KUKA KRL program: MyProgram_293().src

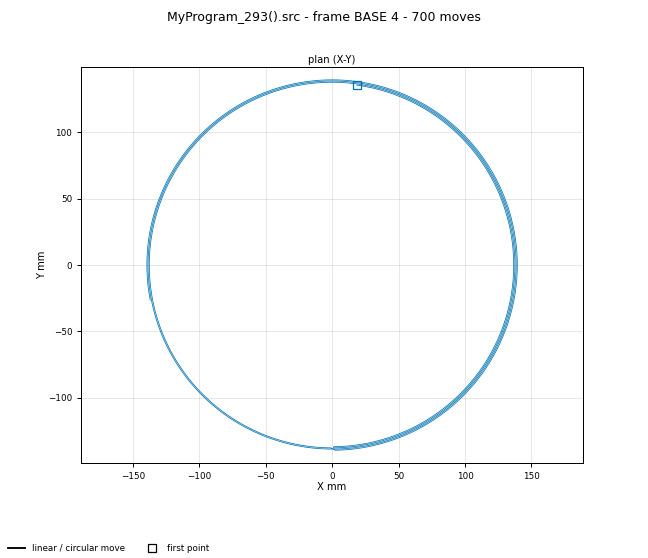
[picture p0: tool path of MyProgram_293().src in frame BASE 4, 700 of 700 moves have a stored position in this frame; points joined in program order, loops and branches not executed]
&ACCESS RVP
&REL 1
&PARAM TEMPLATE = C:\KRC\Roboter\Template\vorgabe
&PARAM EDITMASK = *
DEF MyProgram_293()
; ---- Setting reference (Base) ----
$BASE = BASE_DATA[4]

; --------------------------
; ---- Setting tool (TCP) ----
$TOOL = TOOL_DATA[3]
; --------------------------

$VEL.CP = VEL_APROX_PRINT
Startdeposition()
$VEL.CP = VEL_PRINT
LIN {X 18.5664,Y 135.4056,Z 177,A 82.6594,B 6.5518,C 0.1123,E1 6.5775,E2 369.6797} C_DIS
LIN {X 22.4593,Y 134.8123,Z 177,A 81.1585,B 6.5518,C 0.1109,E1 6.5816,E2 371.162} C_DIS
LIN {X 25.6947,Y 134.2332,Z 177,A 79.7863,B 6.5518,C 0.1116,E1 6.5854,E2 372.533} C_DIS
LIN {X 28.7602,Y 133.61,Z 177,A 78.4781,B 6.5518,C 0.1123,E1 6.589,E2 373.8405} C_DIS
LIN {X 32.2481,Y 132.8114,Z 177,A 76.9941,B 6.5518,C 0.1131,E1 6.593,E2 375.3222} C_DIS
LIN {X 35.7369,Y 131.9163,Z 177,A 75.4178,B 6.5518,C 0.1152,E1 6.5973,E2 376.9062} C_DIS
LIN {X 40.0506,Y 130.6702,Z 177,A 73.6118,B 6.5518,C 0.1156,E1 6.6021,E2 378.7026} C_DIS
LIN {X 43.4189,Y 129.5901,Z 177,A 72.1587,B 6.5517,C 0.1165,E1 6.6059,E2 380.1517} C_DIS
LIN {X 46.8464,Y 128.3916,Z 177,A 70.6202,B 6.5517,C 0.1182,E1 6.61,E2 381.6921} C_DIS
LIN {X 49.9108,Y 127.2313,Z 177,A 69.2422,B 6.5517,C 0.1197,E1 6.6136,E2 383.0704} C_DIS
LIN {X 52.8843,Y 126.0238,Z 177,A 67.9305,B 6.5517,C 0.1207,E1 6.6169,E2 384.3778} C_DIS
LIN {X 56.0642,Y 124.6418,Z 177,A 66.4902,B 6.5516,C 0.1222,E1 6.6206,E2 385.8164} C_DIS
LIN {X 59.3143,Y 123.1288,Z 177,A 64.9808,B 6.5516,C 0.1241,E1 6.6244,E2 387.3264} C_DIS
LIN {X 62.5726,Y 121.5062,Z 177,A 63.4613,B 6.5516,C 0.126,E1 6.6282,E2 388.8452} C_DIS
LIN {X 66.4914,Y 119.4079,Z 177,A 61.5636,B 6.5515,C 0.1291,E1 6.6329,E2 390.747} C_DIS
LIN {X 70.3636,Y 117.1681,Z 177,A 59.6863,B 6.5514,C 0.1319,E1 6.6374,E2 392.6246} C_DIS
LIN {X 74.1474,Y 114.8108,Z 177,A 57.8365,B 6.5514,C 0.1345,E1 6.6418,E2 394.4722} C_DIS
LIN {X 77.7972,Y 112.3696,Z 177,A 56.0558,B 6.5514,C 0.1365,E1 6.6459,E2 396.2457} C_DIS
LIN {X 81.159,Y 109.9661,Z 177,A 54.3535,B 6.5513,C 0.1389,E1 6.6497,E2 397.9445} C_DIS
LIN {X 84.4152,Y 107.4864,Z 177,A 52.6402,B 6.5512,C 0.1419,E1 6.6535,E2 399.6577} C_DIS
LIN {X 88.0221,Y 104.5534,Z 177,A 50.7109,B 6.5512,C 0.1452,E1 6.6576,E2 401.585} C_DIS
LIN {X 91.3809,Y 101.6309,Z 177,A 48.8831,B 6.5511,C 0.1481,E1 6.6614,E2 403.4084} C_DIS
LIN {X 95.3201,Y 97.9461,Z 177,A 46.6989,B 6.551,C 0.1513,E1 6.6659,E2 405.5837} C_DIS
LIN {X 98.313,Y 94.9411,Z 177,A 44.7068,B 6.5508,C 0.1584,E1 6.6698,E2 407.6024} C_DIS
LIN {X 100.5411,Y 92.5782,Z 177,A 43.7698,B 6.5509,C 0.1543,E1 6.6715,E2 408.4878} C_DIS
LIN {X 102.7371,Y 90.1358,Z 177,A 42.1809,B 6.5508,C 0.1608,E1 6.6745,E2 410.1031} C_DIS
LIN {X 105.6039,Y 86.7593,Z 177,A 40.2759,B 6.5506,C 0.1656,E1 6.6779,E2 412.0147} C_DIS
LIN {X 108.5925,Y 82.9874,Z 177,A 38.4354,B 6.5506,C 0.1672,E1 6.681,E2 413.8341} C_DIS
LIN {X 111.0305,Y 79.6965,Z 177,A 36.7303,B 6.5505,C 0.171,E1 6.6838,E2 415.5384} C_DIS
LIN {X 113.4927,Y 76.1495,Z 177,A 34.9398,B 6.5504,C 0.175,E1 6.6866,E2 417.3273} C_DIS
LIN {X 115.869,Y 72.4825,Z 177,A 33.1063,B 6.5503,C 0.1794,E1 6.6894,E2 419.1618} C_DIS
LIN {X 118.1937,Y 68.6259,Z 177,A 31.298,B 6.5502,C 0.1827,E1 6.692,E2 420.9611} C_DIS
LIN {X 120.235,Y 64.9838,Z 177,A 29.5546,B 6.5501,C 0.187,E1 6.6943,E2 422.7045} C_DIS
LIN {X 122.018,Y 61.5673,Z 177,A 28.0806,B 6.5501,C 0.1887,E1 6.6962,E2 424.1618} C_DIS
LIN {X 123.5453,Y 58.4425,Z 177,A 26.6295,B 6.5499,C 0.1923,E1 6.6979,E2 425.6128} C_DIS
LIN {X 125.2833,Y 54.6165,Z 177,A 24.7215,B 6.5497,C 0.1994,E1 6.7001,E2 427.5399} C_DIS
LIN {X 127.4324,Y 49.3935,Z 177,A 22.5717,B 6.5497,C 0.2019,E1 6.7023,E2 429.664} C_DIS
LIN {X 128.7184,Y 45.9402,Z 177,A 21.1087,B 6.5495,C 0.2047,E1 6.7037,E2 431.1179} C_DIS
LIN {X 129.7831,Y 42.8393,Z 177,A 19.728,B 6.5495,C 0.2085,E1 6.7049,E2 432.5002} C_DIS
LIN {X 130.8966,Y 39.3108,Z 177,A 18.2472,B 6.5493,C 0.2115,E1 6.7062,E2 433.9733} C_DIS
LIN {X 131.7436,Y 36.3672,Z 177,A 16.9687,B 6.5493,C 0.215,E1 6.7071,E2 435.2519} C_DIS
LIN {X 132.7743,Y 32.402,Z 177,A 15.2361,B 6.549,C 0.22,E1 6.7083,E2 436.9875} C_DIS
LIN {X 133.655,Y 28.5517,Z 177,A 13.6632,B 6.549,C 0.2232,E1 6.7093,E2 438.5512} C_DIS
LIN {X 134.3809,Y 24.9221,Z 177,A 12.0063,B 6.5487,C 0.2294,E1 6.7101,E2 440.2223} C_DIS
LIN {X 135.1025,Y 20.6444,Z 177,A 10.356,B 6.5487,C 0.2316,E1 6.7109,E2 441.853} C_DIS
LIN {X 135.6098,Y 17.0107,Z 177,A 8.7647,B 6.5485,C 0.2369,E1 6.7115,E2 443.4521} C_DIS
LIN {X 136.0754,Y 12.744,Z 177,A 7.0882,B 6.5483,C 0.2398,E1 6.7119,E2 445.1145} C_DIS
LIN {X 136.5806,Y 4.9707,Z 177,A 3.1417,B 6.5475,C 0.261,E1 6.7125,E2 449.1483} C_DIS
LIN {X 136.6684,Y -0.9178,Z 177,A 1.5135,B 6.5478,C 0.2535,E1 6.7125,E2 450.6738} C_DIS
LIN {X 136.5954,Y -4.5594,Z 177,A -0.5926,B 6.5473,C 0.2679,E1 6.7123,E2 452.8536} C_DIS
LIN {X 136.3436,Y -9.46,Z 177,A -2.4912,B 6.5471,C 0.2711,E1 6.712,E2 454.7342} C_DIS
LIN {X 135.9744,Y -13.7962,Z 177,A -3.8455,B 6.5473,C 0.2681,E1 6.7116,E2 456.0312} C_DIS
LIN {X 135.5357,Y -17.576,Z 177,A -5.43,B 6.5471,C 0.2725,E1 6.7111,E2 457.6157} C_DIS
LIN {X 134.9783,Y -21.4462,Z 177,A -7.0242,B 6.5469,C 0.2764,E1 6.7104,E2 459.2057} C_DIS
LIN {X 134.2054,Y -25.8402,Z 177,A -8.78,B 6.5468,C 0.2797,E1 6.7095,E2 460.9488} C_DIS
LIN {X 133.4372,Y -29.5604,Z 177,A -10.4906,B 6.5465,C 0.2862,E1 6.7085,E2 462.6757} C_DIS
LIN {X 132.2578,Y -34.4551,Z 177,A -12.5264,B 6.5463,C 0.2908,E1 6.7072,E2 464.704} C_DIS
LIN {X 131.2025,Y -38.2708,Z 177,A -14.1081,B 6.5461,C 0.2941,E1 6.706,E2 466.2773} C_DIS
LIN {X 130.0503,Y -42.022,Z 177,A -15.6724,B 6.5461,C 0.2972,E1 6.7047,E2 467.8329} C_DIS
LIN {X 128.5427,Y -46.4275,Z 177,A -17.6099,B 6.5458,C 0.3023,E1 6.7029,E2 469.7704} C_DIS
LIN {X 127.3413,Y -49.6278,Z 177,A -18.9635,B 6.5457,C 0.3048,E1 6.7015,E2 471.1152} C_DIS
LIN {X 125.9129,Y -53.1498,Z 177,A -20.5159,B 6.5455,C 0.3083,E1 6.6999,E2 472.664} C_DIS
LIN {X 124.6312,Y -56.088,Z 177,A -21.8391,B 6.5453,C 0.3115,E1 6.6984,E2 473.9858} C_DIS
LIN {X 123.3542,Y -58.8426,Z 177,A -23.2918,B 6.545,C 0.318,E1 6.6966,E2 475.4624} C_DIS
LIN {X 120.828,Y -63.8703,Z 177,A -25.421,B 6.545,C 0.3201,E1 6.694,E2 477.5647} C_DIS
LIN {X 118.8197,Y -67.5365,Z 177,A -27.2091,B 6.5447,C 0.3252,E1 6.6915,E2 479.3591} C_DIS
LIN {X 116.5896,Y -71.3171,Z 177,A -29.036,B 6.5445,C 0.3296,E1 6.6889,E2 481.1861} C_DIS
LIN {X 114.2108,Y -75.0675,Z 177,A -30.8592,B 6.5443,C 0.3335,E1 6.6861,E2 483.0061} C_DIS
LIN {X 111.7205,Y -78.726,Z 177,A -32.6652,B 6.5441,C 0.3371,E1 6.6833,E2 484.8075} C_DIS
LIN {X 109.1483,Y -82.2551,Z 177,A -34.483,B 6.5439,C 0.3412,E1 6.6802,E2 486.6255} C_DIS
LIN {X 106.402,Y -85.7779,Z 177,A -36.3143,B 6.5437,C 0.3448,E1 6.6771,E2 488.4533} C_DIS
LIN {X 103.4246,Y -89.3456,Z 177,A -38.2127,B 6.5435,C 0.3484,E1 6.6737,E2 490.3471} C_DIS
LIN {X 100.4923,Y -92.6313,Z 177,A -40.0388,B 6.5433,C 0.3521,E1 6.6702,E2 492.1724} C_DIS
LIN {X 97.385,Y -95.893,Z 177,A -41.8836,B 6.5431,C 0.3554,E1 6.6667,E2 494.0133} C_DIS
LIN {X 94.0387,Y -99.1762,Z 177,A -44.0328,B 6.5427,C 0.3625,E1 6.6623,E2 496.1876} C_DIS
LIN {X 91.5951,Y -101.4381,Z 177,A -45.4879,B 6.5425,C 0.3663,E1 6.6592,E2 497.6516} C_DIS
LIN {X 88.7953,Y -103.8978,Z 177,A -46.7251,B 6.5427,C 0.3639,E1 6.6567,E2 498.8488} C_DIS
LIN {X 85.4483,Y -106.6677,Z 177,A -48.5875,B 6.5424,C 0.368,E1 6.6527,E2 500.718} C_DIS
LIN {X 81.8828,Y -109.4283,Z 177,A -50.4029,B 6.5423,C 0.3702,E1 6.6487,E2 502.5255} C_DIS
LIN {X 78.4278,Y -111.9308,Z 177,A -52.2025,B 6.5421,C 0.3736,E1 6.6445,E2 504.3281} C_DIS
LIN {X 74.7223,Y -114.4375,Z 177,A -54.0556,B 6.542,C 0.3763,E1 6.6402,E2 506.1799} C_DIS
LIN {X 70.9075,Y -116.8393,Z 177,A -55.9071,B 6.5418,C 0.3787,E1 6.6359,E2 508.028} C_DIS
LIN {X 67.0797,Y -119.078,Z 177,A -57.7385,B 6.5417,C 0.3811,E1 6.6314,E2 509.8575} C_DIS
LIN {X 63.2452,Y -121.1563,Z 177,A -59.4788,B 6.5417,C 0.3823,E1 6.6272,E2 511.5879} C_DIS
LIN {X 60.1595,Y -122.7177,Z 177,A -60.9304,B 6.5415,C 0.3844,E1 6.6235,E2 513.0408} C_DIS
LIN {X 55.3417,Y -124.965,Z 177,A -63.1051,B 6.5414,C 0.3864,E1 6.618,E2 515.2104} C_DIS
LIN {X 46.6553,Y -128.4605,Z 177,A -66.795,B 6.5414,C 0.3873,E1 6.6085,E2 518.8732} C_DIS
LIN {X 43.9146,Y -129.425,Z 177,A -68.2318,B 6.541,C 0.392,E1 6.6046,E2 520.339} C_DIS
LIN {X 41.2908,Y -130.2839,Z 177,A -69.3344,B 6.541,C 0.3923,E1 6.6017,E2 521.4353} C_DIS
LIN {X 37.4387,Y -131.444,Z 177,A -71.1076,B 6.5408,C 0.3952,E1 6.5969,E2 523.2207} C_DIS
LIN {X 33.4016,Y -132.526,Z 177,A -72.7347,B 6.5408,C 0.3947,E1 6.5926,E2 524.833} C_DIS
LIN {X 30.3416,Y -133.2597,Z 177,A -74.0599,B 6.5408,C 0.3958,E1 6.589,E2 526.1597} C_DIS
LIN {X 27.0594,Y -133.9649,Z 177,A -75.4746,B 6.5408,C 0.3969,E1 6.5851,E2 527.5763} C_DIS
LIN {X 23.3736,Y -134.6587,Z 177,A -77.112,B 6.5406,C 0.3989,E1 6.5806,E2 529.223} C_DIS
LIN {X 16.7281,Y -135.6439,Z 177,A -79.715,B 6.5407,C 0.3972,E1 6.5735,E2 531.8004} C_DIS
LIN {X 12.2421,Y -136.1223,Z 177,A -82.1222,B 6.5402,C 0.4056,E1 6.5666,E2 534.2745} C_DIS
LIN {X 8.4372,Y -136.4098,Z 177,A -83.1352,B 6.5407,C 0.3974,E1 6.564,E2 535.2135} C_DIS
LIN {X 1.4274,Y -136.6648,Z 177,A -86.1789,B 6.5406,C 0.3996,E1 6.5554,E2 538.272} C_DIS
LIN {X 1.4274,Y -136.6648,Z 177,A -86.1789,B 6.5406,C 0.3996,E1 6.5554,E2 538.272} C_DIS
Enddeposition()
LIN {X 0.9977,Y -137.5702,Z 177,A -85.891,B 6.5463,C 0.3964,E1 6.5618,E2 537.955} C_DIS
Startdeposition()
$VEL.CP = VEL_PRINT
LIN {X 3.7285,Y -137.5249,Z 177,A -84.6313,B 6.5464,C 0.3944,E1 6.5654,E2 536.6789} C_DIS
LIN {X 6.8134,Y -137.4065,Z 177,A -83.3451,B 6.5464,C 0.3941,E1 6.569,E2 535.392} C_DIS
LIN {X 10.1117,Y -137.2032,Z 177,A -82.0399,B 6.5464,C 0.3947,E1 6.5726,E2 534.0952} C_DIS
LIN {X 13.0514,Y -136.9548,Z 177,A -80.7476,B 6.5465,C 0.3933,E1 6.5762,E2 532.794} C_DIS
LIN {X 16.3923,Y -136.5952,Z 177,A -79.4157,B 6.5465,C 0.3937,E1 6.5799,E2 531.4702} C_DIS
LIN {X 20.2553,Y -136.0783,Z 177,A -77.7612,B 6.5465,C 0.3924,E1 6.5845,E2 529.8107} C_DIS
LIN {X 23.4383,Y -135.5663,Z 177,A -76.4224,B 6.5466,C 0.3916,E1 6.5882,E2 528.4716} C_DIS
LIN {X 26.6321,Y -134.9752,Z 177,A -75.0021,B 6.5467,C 0.3897,E1 6.5921,E2 527.0416} C_DIS
LIN {X 30.34,Y -134.1882,Z 177,A -73.4718,B 6.5467,C 0.3893,E1 6.5963,E2 525.5165} C_DIS
LIN {X 34.6459,Y -133.1436,Z 177,A -71.6655,B 6.5467,C 0.3884,E1 6.6011,E2 523.7142} C_DIS
LIN {X 37.8556,Y -132.2669,Z 177,A -70.2873,B 6.5469,C 0.3873,E1 6.6048,E2 522.3361} C_DIS
LIN {X 41.2103,Y -131.2594,Z 177,A -68.8943,B 6.5469,C 0.387,E1 6.6085,E2 520.9506} C_DIS
LIN {X 44.2654,Y -130.2618,Z 177,A -67.4751,B 6.547,C 0.3843,E1 6.6123,E2 519.5199} C_DIS
LIN {X 47.4593,Y -129.1324,Z 177,A -66.1069,B 6.547,C 0.3835,E1 6.6159,E2 518.1562} C_DIS
LIN {X 50.6416,Y -127.918,Z 177,A -64.6992,B 6.5472,C 0.382,E1 6.6196,E2 516.7489} C_DIS
LIN {X 54.2347,Y -126.4341,Z 177,A -63.1019,B 6.5472,C 0.3804,E1 6.6237,E2 515.1531} C_DIS
LIN {X 56.9581,Y -125.2331,Z 177,A -61.8648,B 6.5473,C 0.3788,E1 6.6268,E2 513.9156} C_DIS
LIN {X 60.0858,Y -123.7629,Z 177,A -60.439,B 6.5474,C 0.3771,E1 6.6304,E2 512.4904} C_DIS
LIN {X 63.1886,Y -122.2079,Z 177,A -58.8981,B 6.5477,C 0.3735,E1 6.6343,E2 510.9358} C_DIS
LIN {X 67.027,Y -120.1456,Z 177,A -57.1262,B 6.5477,C 0.3716,E1 6.6386,E2 509.168} C_DIS
LIN {X 70.8146,Y -117.9528,Z 177,A -55.3047,B 6.5479,C 0.3688,E1 6.643,E2 507.3453} C_DIS
LIN {X 74.5451,Y -115.6313,Z 177,A -53.4961,B 6.5481,C 0.3661,E1 6.6473,E2 505.5379} C_DIS
LIN {X 78.2897,Y -113.1292,Z 177,A -51.6664,B 6.5482,C 0.3637,E1 6.6515,E2 503.7126} C_DIS
LIN {X 81.8087,Y -110.6115,Z 177,A -49.8837,B 6.5484,C 0.3608,E1 6.6555,E2 501.9309} C_DIS
LIN {X 85.3293,Y -107.9189,Z 177,A -48.04,B 6.5485,C 0.3575,E1 6.6596,E2 500.0858} C_DIS
LIN {X 88.7677,Y -105.1088,Z 177,A -46.24,B 6.5487,C 0.3548,E1 6.6634,E2 498.2906} C_DIS
LIN {X 92.1181,Y -102.1852,Z 177,A -44.3969,B 6.5489,C 0.3512,E1 6.6673,E2 496.4469} C_DIS
LIN {X 95.3794,Y -99.1481,Z 177,A -42.571,B 6.5491,C 0.348,E1 6.671,E2 494.6233} C_DIS
LIN {X 98.533,Y -96.0147,Z 177,A -40.7667,B 6.5492,C 0.3449,E1 6.6745,E2 492.8235} C_DIS
LIN {X 101.5873,Y -92.7771,Z 177,A -38.9249,B 6.5494,C 0.341,E1 6.678,E2 490.9815} C_DIS
LIN {X 104.5331,Y -89.445,Z 177,A -37.1234,B 6.5496,C 0.3378,E1 6.6813,E2 489.1849} C_DIS
LIN {X 107.3661,Y -86.0237,Z 177,A -35.3063,B 6.5498,C 0.3341,E1 6.6845,E2 487.3703} C_DIS
LIN {X 110.0826,Y -82.5191,Z 177,A -33.4933,B 6.55,C 0.3304,E1 6.6876,E2 485.56} C_DIS
LIN {X 112.6788,Y -78.937,Z 177,A -31.6667,B 6.5502,C 0.3263,E1 6.6905,E2 483.7337} C_DIS
LIN {X 115.1518,Y -75.2838,Z 177,A -29.8604,B 6.5504,C 0.3223,E1 6.6933,E2 481.9297} C_DIS
LIN {X 117.4987,Y -71.5655,Z 177,A -28.0881,B 6.5505,C 0.3188,E1 6.6959,E2 480.1634} C_DIS
LIN {X 119.7174,Y -67.7888,Z 177,A -26.2978,B 6.5507,C 0.3148,E1 6.6984,E2 478.3757} C_DIS
LIN {X 121.3987,Y -64.7296,Z 177,A -24.9613,B 6.5508,C 0.3131,E1 6.7002,E2 477.053} C_DIS
LIN {X 122.996,Y -61.6405,Z 177,A -23.5235,B 6.551,C 0.3096,E1 6.702,E2 475.6152} C_DIS
LIN {X 124.6916,Y -58.1293,Z 177,A -22.1099,B 6.551,C 0.309,E1 6.7036,E2 474.2272} C_DIS
LIN {X 126.1301,Y -54.9379,Z 177,A -20.7016,B 6.5511,C 0.306,E1 6.7052,E2 472.8239} C_DIS
LIN {X 127.2787,Y -52.2273,Z 177,A -19.3258,B 6.5514,C 0.3001,E1 6.7067,E2 471.4278} C_DIS
LIN {X 128.5358,Y -49.0521,Z 177,A -17.9343,B 6.5516,C 0.2968,E1 6.7081,E2 470.0389} C_DIS
LIN {X 129.7078,Y -45.8636,Z 177,A -16.5505,B 6.5517,C 0.2935,E1 6.7095,E2 468.6577} C_DIS
LIN {X 130.7947,Y -42.6651,Z 177,A -15.1743,B 6.5519,C 0.2902,E1 6.7107,E2 467.2843} C_DIS
LIN {X 131.7972,Y -39.4598,Z 177,A -13.8072,B 6.552,C 0.2869,E1 6.7118,E2 465.9199} C_DIS
LIN {X 132.7157,Y -36.2508,Z 177,A -12.4483,B 6.5521,C 0.2836,E1 6.7128,E2 464.5637} C_DIS
LIN {X 133.5509,Y -33.0413,Z 177,A -11.0985,B 6.5523,C 0.2802,E1 6.7137,E2 463.2167} C_DIS
LIN {X 134.3357,Y -29.6861,Z 177,A -9.6225,B 6.5525,C 0.2755,E1 6.7146,E2 461.7341} C_DIS
LIN {X 134.9752,Y -26.6321,Z 177,A -8.3075,B 6.5527,C 0.2715,E1 6.7154,E2 460.416} C_DIS
LIN {X 135.5663,Y -23.4383,Z 177,A -7.1048,B 6.5527,C 0.2704,E1 6.7159,E2 459.2314} C_DIS
LIN {X 136.0783,Y -20.2553,Z 177,A -5.7931,B 6.5528,C 0.2671,E1 6.7165,E2 457.9225} C_DIS
LIN {X 136.579,Y -16.528,Z 177,A -4.4655,B 6.5528,C 0.2669,E1 6.717,E2 456.624} C_DIS
LIN {X 136.8703,Y -13.932,Z 177,A -3.201,B 6.5531,C 0.2606,E1 6.7174,E2 455.3361} C_DIS
LIN {X 137.1532,Y -10.7967,Z 177,A -1.9207,B 6.5532,C 0.2574,E1 6.7176,E2 454.0586} C_DIS
LIN {X 137.3629,Y -7.6821,Z 177,A -0.6516,B 6.5533,C 0.2543,E1 6.7179,E2 452.7924} C_DIS
LIN {X 137.5009,Y -4.5903,Z 177,A 0.7505,B 6.5536,C 0.2485,E1 6.718,E2 451.3747} C_DIS
LIN {X 137.5691,Y -1.5235,Z 177,A 1.8807,B 6.5536,C 0.2475,E1 6.718,E2 450.2623} C_DIS
LIN {X 137.5691,Y 1.5235,Z 177,A 3.0967,B 6.5537,C 0.2448,E1 6.718,E2 449.0521} C_DIS
LIN {X 137.5009,Y 4.5903,Z 177,A 4.3491,B 6.5538,C 0.2416,E1 6.718,E2 447.8018} C_DIS
LIN {X 137.3629,Y 7.6821,Z 177,A 5.6126,B 6.5539,C 0.2383,E1 6.7178,E2 446.5406} C_DIS
LIN {X 137.1532,Y 10.7967,Z 177,A 6.9567,B 6.5541,C 0.2339,E1 6.7175,E2 445.1898} C_DIS
LIN {X 136.8703,Y 13.932,Z 177,A 8.172,B 6.5541,C 0.2318,E1 6.7172,E2 443.9857} C_DIS
LIN {X 136.5125,Y 17.0857,Z 177,A 9.4679,B 6.5543,C 0.2285,E1 6.7167,E2 442.6922} C_DIS
LIN {X 136.0783,Y 20.2553,Z 177,A 10.7736,B 6.5544,C 0.2252,E1 6.7162,E2 441.3889} C_DIS
LIN {X 135.4654,Y 24.0017,Z 177,A 12.2904,B 6.5545,C 0.2219,E1 6.7155,E2 439.879} C_DIS
LIN {X 134.9719,Y 26.6483,Z 177,A 13.4166,B 6.5546,C 0.2186,E1 6.7149,E2 438.7514} C_DIS
LIN {X 134.3038,Y 29.834,Z 177,A 14.7514,B 6.5547,C 0.2152,E1 6.7141,E2 437.4184} C_DIS
LIN {X 133.5509,Y 33.0413,Z 177,A 16.1839,B 6.5549,C 0.2104,E1 6.7132,E2 435.9772} C_DIS
LIN {X 132.6126,Y 36.6192,Z 177,A 17.6102,B 6.5549,C 0.2081,E1 6.7121,E2 434.5644} C_DIS
LIN {X 131.7972,Y 39.4598,Z 177,A 18.8138,B 6.5551,C 0.2052,E1 6.7112,E2 433.3635} C_DIS
LIN {X 130.6278,Y 43.1663,Z 177,A 20.3612,B 6.5551,C 0.202,E1 6.7099,E2 431.8239} C_DIS
LIN {X 129.6113,Y 46.1312,Z 177,A 21.5781,B 6.5552,C 0.2001,E1 6.7088,E2 430.6176} C_DIS
LIN {X 128.5358,Y 49.0521,Z 177,A 22.9527,B 6.5554,C 0.1952,E1 6.7074,E2 429.2322} C_DIS
LIN {X 127.2787,Y 52.2273,Z 177,A 24.4355,B 6.5555,C 0.1904,E1 6.7059,E2 427.7409} C_DIS
LIN {X 125.9363,Y 55.386,Z 177,A 25.8381,B 6.5555,C 0.1871,E1 6.7043,E2 426.341} C_DIS
LIN {X 124.5087,Y 58.5249,Z 177,A 27.1595,B 6.5556,C 0.1854,E1 6.7028,E2 425.0333} C_DIS
LIN {X 122.996,Y 61.6405,Z 177,A 28.6123,B 6.5558,C 0.1815,E1 6.701,E2 423.5784} C_DIS
LIN {X 121.059,Y 65.362,Z 177,A 30.3076,B 6.5558,C 0.178,E1 6.6988,E2 421.8888} C_DIS
LIN {X 119.0914,Y 68.8812,Z 177,A 32.0128,B 6.556,C 0.1734,E1 6.6964,E2 420.1795} C_DIS
LIN {X 116.7791,Y 72.7325,Z 177,A 33.8466,B 6.556,C 0.1695,E1 6.6937,E2 418.3495} C_DIS
LIN {X 114.3926,Y 76.4311,Z 177,A 35.6313,B 6.5562,C 0.1659,E1 6.691,E2 416.5701} C_DIS
LIN {X 111.8808,Y 80.0628,Z 177,A 37.4386,B 6.5562,C 0.1622,E1 6.6881,E2 414.766} C_DIS
LIN {X 109.3123,Y 83.5356,Z 177,A 39.2275,B 6.5564,C 0.1582,E1 6.6851,E2 412.9778} C_DIS
LIN {X 106.4935,Y 87.1006,Z 177,A 41.0684,B 6.5564,C 0.1549,E1 6.6819,E2 411.1427} C_DIS
LIN {X 103.5973,Y 90.5261,Z 177,A 42.8987,B 6.5565,C 0.1515,E1 6.6786,E2 409.3166} C_DIS
LIN {X 100.6447,Y 93.7977,Z 177,A 44.7123,B 6.5565,C 0.148,E1 6.6751,E2 407.5052} C_DIS
LIN {X 97.5157,Y 97.0468,Z 177,A 46.5511,B 6.5567,C 0.1448,E1 6.6716,E2 405.6709} C_DIS
LIN {X 94.447,Y 100.0357,Z 177,A 48.339,B 6.5567,C 0.1412,E1 6.668,E2 403.8821} C_DIS
LIN {X 91.0815,Y 103.1093,Z 177,A 50.1885,B 6.5568,C 0.1383,E1 6.6641,E2 402.0383} C_DIS
LIN {X 87.7864,Y 105.9289,Z 177,A 51.9892,B 6.5568,C 0.1351,E1 6.6603,E2 400.238} C_DIS
LIN {X 84.2772,Y 108.7416,Z 177,A 53.8245,B 6.5569,C 0.1324,E1 6.6563,E2 398.4071} C_DIS
LIN {X 80.6195,Y 111.4804,Z 177,A 55.6771,B 6.5569,C 0.13,E1 6.6521,E2 396.5606} C_DIS
LIN {X 77.0741,Y 113.9603,Z 177,A 57.4712,B 6.557,C 0.1272,E1 6.648,E2 394.7673} C_DIS
LIN {X 73.3868,Y 116.3691,Z 177,A 59.2823,B 6.557,C 0.1247,E1 6.6437,E2 392.959} C_DIS
LIN {X 69.7298,Y 118.5966,Z 177,A 61.0643,B 6.5571,C 0.1221,E1 6.6395,E2 391.1772} C_DIS
LIN {X 65.9269,Y 120.7519,Z 177,A 62.8145,B 6.5571,C 0.1206,E1 6.6352,E2 389.4357} C_DIS
LIN {X 63.1886,Y 122.2079,Z 177,A 64.1332,B 6.5571,C 0.1185,E1 6.6319,E2 388.1137} C_DIS
LIN {X 60.0858,Y 123.7629,Z 177,A 65.4966,B 6.5571,C 0.1179,E1 6.6285,E2 386.7605} C_DIS
LIN {X 56.9581,Y 125.2331,Z 177,A 67.053,B 6.5573,C 0.1144,E1 6.6246,E2 385.1897} C_DIS
LIN {X 53.4574,Y 126.765,Z 177,A 68.3572,B 6.5573,C 0.117,E1 6.6213,E2 383.9212} C_DIS
LIN {X 50.6416,Y 127.918,Z 177,A 69.7521,B 6.5573,C 0.1137,E1 6.6177,E2 382.5107} C_DIS
LIN {X 47.4593,Y 129.1324,Z 177,A 71.2995,B 6.5573,C 0.1102,E1 6.6136,E2 380.9475} C_DIS
LIN {X 43.8871,Y 130.3878,Z 177,A 72.6905,B 6.5573,C 0.1116,E1 6.6099,E2 379.5797} C_DIS
LIN {X 40.8564,Y 131.3697,Z 177,A 73.9579,B 6.5573,C 0.1113,E1 6.6066,E2 378.32} C_DIS
LIN {X 37.8556,Y 132.2669,Z 177,A 75.332,B 6.5573,C 0.1092,E1 6.6029,E2 376.9376} C_DIS
LIN {X 34.3144,Y 133.2278,Z 177,A 76.7233,B 6.5573,C 0.1101,E1 6.5992,E2 375.5634} C_DIS
LIN {X 31.4372,Y 133.9376,Z 177,A 78.1706,B 6.5573,C 0.1061,E1 6.5952,E2 374.0902} C_DIS
LIN {X 28.2322,Y 134.6496,Z 177,A 79.4332,B 6.5573,C 0.1068,E1 6.5918,E2 372.8408} C_DIS
LIN {X 24.5213,Y 135.3725,Z 177,A 80.9678,B 6.5573,C 0.1065,E1 6.5876,E2 371.3115} C_DIS
LIN {X 21.2848,Y 135.9189,Z 177,A 82.3883,B 6.5574,C 0.1051,E1 6.5836,E2 369.8849} C_DIS
LIN {X 17.0857,Y 136.5125,Z 177,A 84.1163,B 6.5574,C 0.105,E1 6.5789,E2 368.1623} C_DIS
LIN {X 13.932,Y 136.8703,Z 177,A 85.4324,B 6.5574,C 0.1046,E1 6.5752,E2 366.8474} C_DIS
LIN {X 10.7967,Y 137.1532,Z 177,A 86.7385,B 6.5574,C 0.1043,E1 6.5716,E2 365.5424} C_DIS
LIN {X 7.6821,Y 137.3629,Z 177,A 88.0337,B 6.5574,C 0.1042,E1 6.568,E2 364.2482} C_DIS
LIN {X 4.5903,Y 137.5009,Z 177,A 89.3189,B 6.5574,C 0.1041,E1 6.5644,E2 362.9641} C_DIS
LIN {X 1.5235,Y 137.5691,Z 177,A 90.5934,B 6.5574,C 0.1041,E1 6.5608,E2 361.6905} C_DIS
LIN {X -1.5235,Y 137.5691,Z 177,A 91.8634,B 6.5574,C 0.104,E1 6.5573,E2 360.4209} C_DIS
LIN {X -4.5903,Y 137.5009,Z 177,A 93.2485,B 6.5574,C 0.1026,E1 6.5534,E2 359.0231} C_DIS
LIN {X -7.6821,Y 137.3629,Z 177,A 94.4372,B 6.5574,C 0.1041,E1 6.5501,E2 357.8475} C_DIS
LIN {X -10.7967,Y 137.1532,Z 177,A 95.7417,B 6.5574,C 0.1043,E1 6.5465,E2 356.5431} C_DIS
LIN {X -13.932,Y 136.8703,Z 177,A 97.0578,B 6.5574,C 0.1046,E1 6.5428,E2 355.227} C_DIS
LIN {X -17.0857,Y 136.5125,Z 177,A 98.5408,B 6.5574,C 0.1028,E1 6.5386,E2 353.7248} C_DIS
LIN {X -20.2553,Y 136.0783,Z 177,A 99.7241,B 6.5574,C 0.1054,E1 6.5354,E2 352.5607} C_DIS
LIN {X -23.4383,Y 135.5663,Z 177,A 101.0738,B 6.5574,C 0.1059,E1 6.5317,E2 351.2108} C_DIS
LIN {X -26.6321,Y 134.9752,Z 177,A 102.4344,B 6.5574,C 0.1065,E1 6.528,E2 349.8501} C_DIS
LIN {X -29.834,Y 134.3038,Z 177,A 103.9,B 6.5574,C 0.1059,E1 6.5239,E2 348.3726} C_DIS
LIN {X -33.162,Y 133.5203,Z 177,A 105.1919,B 6.5574,C 0.1086,E1 6.5205,E2 347.0978} C_DIS
LIN {X -36.2508,Y 132.7157,Z 177,A 106.5772,B 6.5574,C 0.1088,E1 6.5167,E2 345.7065} C_DIS
LIN {X -39.4598,Y 131.7972,Z 177,A 108.0792,B 6.5574,C 0.1085,E1 6.5127,E2 344.1916} C_DIS
LIN {X -43.2174,Y 130.6108,Z 177,A 109.4149,B 6.5573,C 0.1139,E1 6.5092,E2 342.8946} C_DIS
LIN {X -45.8636,Y 129.7078,Z 177,A 110.8068,B 6.5573,C 0.112,E1 6.5055,E2 341.4755} C_DIS
LIN {X -49.5378,Y 128.347,Z 177,A 112.2585,B 6.5573,C 0.116,E1 6.5017,E2 340.0471} C_DIS
LIN {X -52.2273,Y 127.2787,Z 177,A 113.6702,B 6.5573,C 0.1146,E1 6.498,E2 338.6108} C_DIS
LIN {X -55.386,Y 125.9363,Z 177,A 115.2271,B 6.5573,C 0.1146,E1 6.494,E2 337.0392} C_DIS
LIN {X -58.7225,Y 124.4143,Z 177,A 116.5749,B 6.5572,C 0.1187,E1 6.4906,E2 335.7147} C_DIS
LIN {X -61.6405,Y 122.996,Z 177,A 118.0229,B 6.5572,C 0.1191,E1 6.487,E2 334.2559} C_DIS
LIN {X -65.1602,Y 121.1674,Z 177,A 119.7489,B 6.5572,C 0.1204,E1 6.4827,E2 332.5219} C_DIS
LIN {X -68.8897,Y 119.0865,Z 177,A 121.5678,B 6.5572,C 0.1224,E1 6.4783,E2 330.6994} C_DIS
LIN {X -72.7325,Y 116.7791,Z 177,A 123.4391,B 6.5571,C 0.1251,E1 6.4738,E2 328.829} C_DIS
LIN {X -76.4311,Y 114.3926,Z 177,A 125.2962,B 6.5571,C 0.1277,E1 6.4695,E2 326.9704} C_DIS
LIN {X -80.0628,Y 111.8808,Z 177,A 127.1602,B 6.557,C 0.1304,E1 6.4652,E2 325.1049} C_DIS
LIN {X -83.5356,Y 109.3123,Z 177,A 129.0056,B 6.557,C 0.1329,E1 6.4611,E2 323.2553} C_DIS
LIN {X -87.1006,Y 106.4935,Z 177,A 130.9105,B 6.5568,C 0.1361,E1 6.4569,E2 321.3504} C_DIS
LIN {X -90.5652,Y 103.5632,Z 177,A 132.8063,B 6.5568,C 0.1396,E1 6.4529,E2 319.4555} C_DIS
LIN {X -93.7977,Y 100.6447,Z 177,A 134.665,B 6.5568,C 0.1426,E1 6.4491,E2 317.5929} C_DIS
LIN {X -97.0046,Y 97.5576,Z 177,A 136.5483,B 6.5566,C 0.1459,E1 6.4453,E2 315.7076} C_DIS
LIN {X -100.0357,Y 94.447,Z 177,A 138.4079,B 6.5566,C 0.149,E1 6.4417,E2 313.8432} C_DIS
LIN {X -103.1093,Y 91.0815,Z 177,A 140.3166,B 6.5565,C 0.153,E1 6.4382,E2 311.935} C_DIS
LIN {X -105.9872,Y 87.7159,Z 177,A 142.2105,B 6.5564,C 0.1564,E1 6.4348,E2 310.0366} C_DIS
LIN {X -108.7846,Y 84.2216,Z 177,A 144.0854,B 6.5563,C 0.1605,E1 6.4315,E2 308.162} C_DIS
LIN {X -111.3637,Y 80.7806,Z 177,A 145.9335,B 6.5563,C 0.164,E1 6.4284,E2 306.3085} C_DIS
LIN {X -113.9603,Y 77.0741,Z 177,A 147.8313,B 6.5561,C 0.1683,E1 6.4254,E2 304.4107} C_DIS
LIN {X -116.3691,Y 73.3868,Z 177,A 149.6996,B 6.556,C 0.1723,E1 6.4226,E2 302.54} C_DIS
LIN {X -118.5966,Y 69.7298,Z 177,A 151.5374,B 6.5559,C 0.1761,E1 6.42,E2 300.697} C_DIS
LIN {X -120.7519,Y 65.9269,Z 177,A 153.2175,B 6.5557,C 0.1823,E1 6.4177,E2 299.0361} C_DIS
LIN {X -122.2079,Y 63.1886,Z 177,A 154.6326,B 6.5557,C 0.1841,E1 6.4159,E2 297.6068} C_DIS
LIN {X -123.7629,Y 60.0858,Z 177,A 156.1063,B 6.5556,C 0.1875,E1 6.414,E2 296.1309} C_DIS
LIN {X -125.3395,Y 56.7204,Z 177,A 157.5862,B 6.5554,C 0.1924,E1 6.4123,E2 294.6609} C_DIS
LIN {X -126.6787,Y 53.6641,Z 177,A 159.0427,B 6.5554,C 0.1953,E1 6.4107,E2 293.1973} C_DIS
LIN {X -127.918,Y 50.6416,Z 177,A 160.6076,B 6.5554,C 0.1966,E1 6.409,E2 291.6081} C_DIS
LIN {X -129.1324,Y 47.4593,Z 177,A 161.9374,B 6.5552,C 0.2014,E1 6.4078,E2 290.2908} C_DIS
LIN {X -130.2618,Y 44.2654,Z 177,A 163.3767,B 6.5551,C 0.2049,E1 6.4064,E2 288.8493} C_DIS
LIN {X -131.4648,Y 40.5458,Z 177,A 164.9089,B 6.5549,C 0.2104,E1 6.4052,E2 287.3304} C_DIS
LIN {X -132.2669,Y 37.8556,Z 177,A 166.2316,B 6.5549,C 0.2119,E1 6.4041,E2 285.9896} C_DIS
LIN {X -133.1436,Y 34.6459,Z 177,A 167.6459,B 6.5547,C 0.2155,E1 6.4031,E2 284.573} C_DIS
LIN {X -133.9376,Y 31.4372,Z 177,A 169.1959,B 6.5547,C 0.2173,E1 6.4021,E2 283.0024} C_DIS
LIN {X -134.6496,Y 28.2322,Z 177,A 170.4466,B 6.5545,C 0.2225,E1 6.4013,E2 281.7677} C_DIS
LIN {X -135.2807,Y 25.034,Z 177,A 171.8326,B 6.5544,C 0.226,E1 6.4006,E2 280.3793} C_DIS
LIN {X -135.9049,Y 21.3746,Z 177,A 173.4431,B 6.5542,C 0.2297,E1 6.3999,E2 278.7619} C_DIS
LIN {X -136.349,Y 18.3326,Z 177,A 174.6502,B 6.5541,C 0.2341,E1 6.3994,E2 277.5652} C_DIS
LIN {X -136.7646,Y 14.9136,Z 177,A 175.9567,B 6.5539,C 0.2396,E1 6.399,E2 276.276} C_DIS
LIN {X -137.021,Y 12.3619,Z 177,A 177.2728,B 6.5539,C 0.2399,E1 6.3986,E2 274.9297} C_DIS
LIN {X -137.2671,Y 9.2367,Z 177,A 178.6057,B 6.5538,C 0.2433,E1 6.3984,E2 273.5945} C_DIS
LIN {X -137.4619,Y 5.5906,Z 177,A -179.7872,B 6.5536,C 0.2467,E1 6.3982,E2 271.9777} C_DIS
LIN {X -137.562,Y 1.9459,Z 177,A -178.2219,B 6.5535,C 0.2505,E1 6.3981,E2 270.4077} C_DIS
LIN {X -137.5691,Y -1.5235,Z 177,A -176.8133,B 6.5533,C 0.2551,E1 6.3981,E2 269.0049} C_DIS
LIN {X -137.5009,Y -4.5903,Z 177,A -175.5038,B 6.5532,C 0.2584,E1 6.3981,E2 267.6924} C_DIS
LIN {X -137.3466,Y -7.9456,Z 177,A -174.0181,B 6.5531,C 0.2614,E1 6.3984,E2 266.1968} C_DIS
LIN {X -137.0951,Y -11.4841,Z 177,A -172.5555,B 6.5529,C 0.2658,E1 6.3987,E2 264.7373} C_DIS
LIN {X -136.7008,Y -15.5067,Z 177,A -170.8319,B 6.5527,C 0.2701,E1 6.3992,E2 263.0099} C_DIS
LIN {X -136.305,Y -18.6686,Z 177,A -169.3401,B 6.5527,C 0.272,E1 6.3998,E2 261.4982} C_DIS
LIN {X -135.8097,Y -21.9792,Z 177,A -168.0541,B 6.5524,C 0.2771,E1 6.4003,E2 260.2269} C_DIS
LIN {X -135.2666,Y -25.1075,Z 177,A -166.7189,B 6.5523,C 0.2807,E1 6.401,E2 258.891} C_DIS
LIN {X -134.6381,Y -28.2854,Z 177,A -165.2941,B 6.5521,C 0.2836,E1 6.4018,E2 257.4576} C_DIS
LIN {X -133.9031,Y -31.5804,Z 177,A -163.9253,B 6.552,C 0.2879,E1 6.4026,E2 256.0944} C_DIS
LIN {X -133.1436,Y -34.6459,Z 177,A -162.5234,B 6.5518,C 0.2906,E1 6.4036,E2 254.6825} C_DIS
LIN {X -132.2669,Y -37.8556,Z 177,A -161.1054,B 6.5517,C 0.294,E1 6.4047,E2 253.2613} C_DIS
LIN {X -131.1661,Y -41.5025,Z 177,A -159.4634,B 6.5515,C 0.2976,E1 6.406,E2 251.6132} C_DIS
LIN {X -130.2618,Y -44.2654,Z 177,A -158.2363,B 6.5514,C 0.3007,E1 6.4071,E2 250.3848} C_DIS
LIN {X -129.1324,Y -47.4593,Z 177,A -156.8016,B 6.5512,C 0.3042,E1 6.4085,E2 248.948} C_DIS
LIN {X -127.918,Y -50.6416,Z 177,A -155.3516,B 6.5511,C 0.3076,E1 6.41,E2 247.4949} C_DIS
LIN {X -126.6136,Y -53.8195,Z 177,A -153.7817,B 6.551,C 0.3097,E1 6.4117,E2 245.9079} C_DIS
LIN {X -125.2331,Y -56.9581,Z 177,A -152.4309,B 6.5508,C 0.3143,E1 6.4132,E2 244.5678} C_DIS
LIN {X -123.6546,Y -60.3054,Z 177,A -150.8304,B 6.5506,C 0.3175,E1 6.4151,E2 242.9606} C_DIS
LIN {X -122.1878,Y -63.2268,Z 177,A -149.3733,B 6.5505,C 0.3198,E1 6.417,E2 241.4919} C_DIS
LIN {X -120.1456,Y -67.027,Z 177,A -147.5445,B 6.5503,C 0.3239,E1 6.4195,E2 239.66} C_DIS
LIN {X -117.9528,Y -70.8146,Z 177,A -145.6656,B 6.5501,C 0.3276,E1 6.4222,E2 237.7747} C_DIS
LIN {X -115.6313,Y -74.5451,Z 177,A -143.7998,B 6.5499,C 0.3315,E1 6.425,E2 235.9051} C_DIS
LIN {X -113.1833,Y -78.2119,Z 177,A -141.9285,B 6.5497,C 0.3353,E1 6.4279,E2 234.0301} C_DIS
LIN {X -110.6081,Y -81.8133,Z 177,A -140.0715,B 6.5495,C 0.3393,E1 6.431,E2 232.1721} C_DIS
LIN {X -107.9189,Y -85.3293,Z 177,A -138.1739,B 6.5493,C 0.3427,E1 6.4342,E2 230.2682} C_DIS
LIN {X -105.1088,Y -88.7677,Z 177,A -136.3063,B 6.5491,C 0.3465,E1 6.4376,E2 228.3989} C_DIS
LIN {X -102.1852,Y -92.1181,Z 177,A -134.4099,B 6.549,C 0.3498,E1 6.4411,E2 226.4973} C_DIS
LIN {X -99.1003,Y -95.4288,Z 177,A -132.5137,B 6.5488,C 0.3534,E1 6.4447,E2 224.6002} C_DIS
LIN {X -96.0147,Y -98.533,Z 177,A -130.6639,B 6.5486,C 0.3566,E1 6.4484,E2 222.7473} C_DIS
LIN {X -92.7771,Y -101.5873,Z 177,A -128.7634,B 6.5484,C 0.3595,E1 6.4523,E2 220.8411} C_DIS
LIN {X -89.445,Y -104.5331,Z 177,A -126.9049,B 6.5483,C 0.3627,E1 6.4562,E2 218.9821} C_DIS
LIN {X -86.0237,Y -107.3661,Z 177,A -125.0304,B 6.5481,C 0.3656,E1 6.4603,E2 217.1048} C_DIS
LIN {X -82.5191,Y -110.0826,Z 177,A -123.1606,B 6.5479,C 0.3683,E1 6.4645,E2 215.2323} C_DIS
LIN {X -78.937,Y -112.6788,Z 177,A -121.2772,B 6.5479,C 0.3707,E1 6.4688,E2 213.3437} C_DIS
LIN {X -75.2838,Y -115.1518,Z 177,A -119.4197,B 6.5477,C 0.3732,E1 6.4731,E2 211.4837} C_DIS
LIN {X -71.5655,Y -117.4987,Z 177,A -117.5888,B 6.5475,C 0.3758,E1 6.4774,E2 209.653} C_DIS
LIN {X -67.7888,Y -119.7174,Z 177,A -115.7473,B 6.5474,C 0.378,E1 6.4819,E2 207.8092} C_DIS
LIN {X -64.7296,Y -121.3987,Z 177,A -114.368,B 6.5472,C 0.3808,E1 6.4853,E2 206.4395} C_DIS
LIN {X -61.6405,Y -122.996,Z 177,A -112.9075,B 6.5472,C 0.3824,E1 6.4889,E2 204.9773} C_DIS
LIN {X -58.3221,Y -124.6024,Z 177,A -111.3031,B 6.5471,C 0.3832,E1 6.493,E2 203.3638} C_DIS
LIN {X -55.386,Y -125.9363,Z 177,A -110.007,B 6.547,C 0.3852,E1 6.4963,E2 202.0738} C_DIS
LIN {X -52.2273,Y -127.2787,Z 177,A -108.5681,B 6.547,C 0.3865,E1 6.5,E2 200.6335} C_DIS
LIN {X -49.0521,Y -128.5358,Z 177,A -107.1372,B 6.5468,C 0.3877,E1 6.5037,E2 199.2013} C_DIS
LIN {X -45.8636,Y -129.7078,Z 177,A -105.6314,B 6.5468,C 0.3877,E1 6.5077,E2 197.6835} C_DIS
LIN {X -42.6651,Y -130.7947,Z 177,A -104.3005,B 6.5468,C 0.3898,E1 6.5112,E2 196.3622} C_DIS
LIN {X -39.4598,Y -131.7972,Z 177,A -102.7594,B 6.5468,C 0.3889,E1 6.5154,E2 194.8022} C_DIS
LIN {X -36.2508,Y -132.7157,Z 177,A -101.5009,B 6.5466,C 0.3916,E1 6.5187,E2 193.5605} C_DIS
LIN {X -32.7156,Y -133.6294,Z 177,A -100.0995,B 6.5464,C 0.3942,E1 6.5225,E2 192.1742} C_DIS
LIN {X -29.834,Y -134.3038,Z 177,A -98.7397,B 6.5465,C 0.393,E1 6.5262,E2 190.7976} C_DIS
LIN {X -26.2355,Y -135.051,Z 177,A -97.2345,B 6.5465,C 0.3941,E1 6.5303,E2 189.2952} C_DIS
LIN {X -23.4383,Y -135.5663,Z 177,A -96.0201,B 6.5465,C 0.3941,E1 6.5337,E2 188.0766} C_DIS
LIN {X -20.2553,Y -136.0783,Z 177,A -94.6762,B 6.5465,C 0.3945,E1 6.5374,E2 186.732} C_DIS
LIN {X -17.0857,Y -136.5125,Z 177,A -93.3435,B 6.5465,C 0.3948,E1 6.5411,E2 185.3989} C_DIS
LIN {X -13.4584,Y -136.9157,Z 177,A -91.889,B 6.5463,C 0.3961,E1 6.5451,E2 183.9522} C_DIS
LIN {X -10.7967,Y -137.1532,Z 177,A -90.7123,B 6.5463,C 0.3953,E1 6.5484,E2 182.7668} C_DIS
LIN {X -7.6821,Y -137.3629,Z 177,A -89.4146,B 6.5463,C 0.3953,E1 6.552,E2 181.4688} C_DIS
LIN {X -4.5903,Y -137.5009,Z 177,A -88.1282,B 6.5463,C 0.3953,E1 6.5556,E2 180.1823} C_DIS
LIN {X -0.9625,Y -137.5722,Z 177,A -86.5969,B 6.5464,C 0.395,E1 6.5599,E2 178.6476} C_DIS
LIN {X -0.9625,Y -137.5722,Z 177,A -86.5969,B 6.5464,C 0.395,E1 6.5599,E2 178.6476} C_DIS
Enddeposition()
LIN {X 0.9981,Y -138.4764,Z 177,A -86.4026,B 6.5501,C 0.4079,E1 6.5646,E2 178.5654} C_DIS
Startdeposition()
$VEL.CP = VEL_PRINT
LIN {X -3.0078,Y -138.4493,Z 177,A -88.0923,B 6.5501,C 0.4085,E1 6.5599,E2 180.2601} C_DIS
LIN {X -6.7878,Y -138.3137,Z 177,A -89.6359,B 6.5501,C 0.4082,E1 6.5556,E2 181.8016} C_DIS
LIN {X -10.9292,Y -138.05,Z 177,A -91.4602,B 6.5501,C 0.4096,E1 6.5505,E2 183.6406} C_DIS
LIN {X -15.346,Y -137.6281,Z 177,A -93.2446,B 6.5501,C 0.4086,E1 6.5455,E2 185.4189} C_DIS
LIN {X -19.2919,Y -137.1299,Z 177,A -94.8237,B 6.5501,C 0.4072,E1 6.5412,E2 186.99} C_DIS
LIN {X -26.7728,Y -135.8695,Z 177,A -98.7733,B 6.5495,C 0.4175,E1 6.5301,E2 191.045} C_DIS
LIN {X -32.7318,Y -134.5562,Z 177,A -100.4793,B 6.5503,C 0.4046,E1 6.5257,E2 192.6463} C_DIS
LIN {X -35.4341,Y -133.8698,Z 177,A -101.801,B 6.5503,C 0.4063,E1 6.5221,E2 193.9902} C_DIS
LIN {X -39.9608,Y -132.59,Z 177,A -103.6606,B 6.5503,C 0.4037,E1 6.5171,E2 195.8389} C_DIS
LIN {X -43.4083,Y -131.5009,Z 177,A -105.1162,B 6.5505,C 0.402,E1 6.5133,E2 197.2896} C_DIS
LIN {X -46.3462,Y -130.4956,Z 177,A -106.4862,B 6.5505,C 0.4021,E1 6.5096,E2 198.6709} C_DIS
LIN {X -49.7946,Y -129.2179,Z 177,A -107.8775,B 6.5507,C 0.399,E1 6.506,E2 200.0455} C_DIS
LIN {X -53.118,Y -127.8873,Z 177,A -109.4476,B 6.5507,C 0.3987,E1 6.5019,E2 201.6273} C_DIS
LIN {X -58.4948,Y -125.5194,Z 177,A -111.8597,B 6.5509,C 0.3959,E1 6.4958,E2 204.0373} C_DIS
LIN {X -65.1511,Y -122.1993,Z 177,A -115.0963,B 6.5509,C 0.3944,E1 6.4877,E2 207.2947} C_DIS
LIN {X -69.1025,Y -120.0087,Z 177,A -117.0004,B 6.5511,C 0.3924,E1 6.483,E2 209.2032} C_DIS
LIN {X -72.9928,Y -117.6828,Z 177,A -118.6882,B 6.5514,C 0.3873,E1 6.4791,E2 210.8667} C_DIS
LIN {X -76.263,Y -115.5903,Z 177,A -120.4737,B 6.5514,C 0.3873,E1 6.4748,E2 212.6753} C_DIS
LIN {X -79.1301,Y -113.6467,Z 177,A -122.4177,B 6.5511,C 0.3917,E1 6.4702,E2 214.6847} C_DIS
LIN {X -83.0708,Y -110.7997,Z 177,A -124.0097,B 6.5516,C 0.383,E1 6.4668,E2 216.2228} C_DIS
LIN {X -86.678,Y -108.0008,Z 177,A -125.9188,B 6.5518,C 0.3801,E1 6.4626,E2 218.1342} C_DIS
LIN {X -90.1572,Y -105.1138,Z 177,A -127.8165,B 6.552,C 0.3771,E1 6.4585,E2 220.035} C_DIS
LIN {X -93.6596,Y -102.005,Z 177,A -129.7253,B 6.5522,C 0.3732,E1 6.4546,E2 221.9397} C_DIS
LIN {X -96.7392,Y -99.0897,Z 177,A -131.5684,B 6.5523,C 0.371,E1 6.4508,E2 223.7938} C_DIS
LIN {X -100.0269,Y -95.7694,Z 177,A -133.4882,B 6.5525,C 0.367,E1 6.4471,E2 225.7113} C_DIS
LIN {X -102.9741,Y -92.5935,Z 177,A -135.3467,B 6.5527,C 0.3641,E1 6.4436,E2 227.5778} C_DIS
LIN {X -106.0479,Y -89.0561,Z 177,A -137.2819,B 6.5529,C 0.36,E1 6.4401,E2 229.5118} C_DIS
LIN {X -108.887,Y -85.5615,Z 177,A -139.1805,B 6.5531,C 0.3564,E1 6.4368,E2 231.4143} C_DIS
LIN {X -111.6609,Y -81.9085,Z 177,A -141.1068,B 6.5533,C 0.3525,E1 6.4335,E2 233.3436} C_DIS
LIN {X -114.3553,Y -78.1032,Z 177,A -142.9443,B 6.5536,C 0.3469,E1 6.4306,E2 235.1686} C_DIS
LIN {X -116.3046,Y -75.1697,Z 177,A -144.5846,B 6.5536,C 0.3457,E1 6.4281,E2 236.8316} C_DIS
LIN {X -118.7268,Y -71.283,Z 177,A -146.5289,B 6.5539,C 0.3418,E1 6.4252,E2 238.7814} C_DIS
LIN {X -120.9843,Y -67.38,Z 177,A -148.6344,B 6.5539,C 0.34,E1 6.4223,E2 240.9164} C_DIS
LIN {X -122.5546,Y -64.4744,Z 177,A -149.6516,B 6.5544,C 0.3325,E1 6.421,E2 241.8884} C_DIS
LIN {X -124.0772,Y -61.4939,Z 177,A -151.1156,B 6.5545,C 0.3299,E1 6.4192,E2 243.3618} C_DIS
LIN {X -125.4452,Y -58.6553,Z 177,A -152.5459,B 6.5545,C 0.3281,E1 6.4174,E2 244.8075} C_DIS
LIN {X -126.9783,Y -55.2559,Z 177,A -153.9954,B 6.5548,C 0.323,E1 6.4158,E2 246.2443} C_DIS
LIN {X -128.3219,Y -52.0595,Z 177,A -155.4825,B 6.555,C 0.3199,E1 6.4142,E2 247.7372} C_DIS
LIN {X -129.6288,Y -48.7135,Z 177,A -156.789,B 6.5553,C 0.3139,E1 6.4129,E2 249.02} C_DIS
LIN {X -131.0291,Y -44.8143,Z 177,A -158.8788,B 6.5553,C 0.3136,E1 6.411,E2 251.1565} C_DIS
LIN {X -132.3417,Y -40.7721,Z 177,A -160.6063,B 6.5555,C 0.3085,E1 6.4095,E2 252.8789} C_DIS
LIN {X -133.3485,Y -37.3475,Z 177,A -162.0813,B 6.5557,C 0.3044,E1 6.4084,E2 254.3527} C_DIS
LIN {X -134.3232,Y -33.6762,Z 177,A -163.6995,B 6.5559,C 0.3006,E1 6.4072,E2 255.9758} C_DIS
LIN {X -135.2773,Y -29.6119,Z 177,A -165.4589,B 6.5561,C 0.2962,E1 6.4061,E2 257.738} C_DIS
LIN {X -136.0021,Y -26.0788,Z 177,A -166.9636,B 6.5563,C 0.2922,E1 6.4053,E2 259.2432} C_DIS
LIN {X -136.6455,Y -22.4679,Z 177,A -168.5066,B 6.5565,C 0.2882,E1 6.4046,E2 260.7884} C_DIS
LIN {X -137.2204,Y -18.6468,Z 177,A -170.1914,B 6.5566,C 0.2847,E1 6.4039,E2 262.4829} C_DIS
LIN {X -137.5991,Y -15.6127,Z 177,A -171.3931,B 6.5568,C 0.2804,E1 6.4035,E2 263.6756} C_DIS
LIN {X -137.977,Y -11.7932,Z 177,A -173.0703,B 6.5569,C 0.2769,E1 6.4031,E2 265.3628} C_DIS
LIN {X -138.2481,Y -8.0277,Z 177,A -174.6924,B 6.5571,C 0.2731,E1 6.4028,E2 266.9913} C_DIS
LIN {X -138.405,Y -4.6165,Z 177,A -176.0449,B 6.5573,C 0.2684,E1 6.4026,E2 268.3351} C_DIS
LIN {X -138.4764,Y -1.1527,Z 177,A -177.7239,B 6.5573,C 0.267,E1 6.4026,E2 270.0438} C_DIS
LIN {X -138.4339,Y 3.5886,Z 177,A -179.5368,B 6.5576,C 0.2597,E1 6.4026,E2 271.8363} C_DIS
LIN {X -138.3179,Y 6.7056,Z 177,A 179.0871,B 6.5578,C 0.257,E1 6.4028,E2 273.2221} C_DIS
LIN {X -138.0944,Y 10.3307,Z 177,A 177.3477,B 6.5578,C 0.2553,E1 6.4032,E2 274.9898} C_DIS
LIN {X -137.6019,Y 15.5893,Z 177,A 175.2219,B 6.5581,C 0.2484,E1 6.4038,E2 277.1064} C_DIS
LIN {X -137.0894,Y 19.5757,Z 177,A 173.6397,B 6.5583,C 0.2428,E1 6.4044,E2 278.677} C_DIS
LIN {X -136.4702,Y 23.5181,Z 177,A 171.9727,B 6.5585,C 0.2383,E1 6.4051,E2 280.3446} C_DIS
LIN {X -135.4849,Y 28.6504,Z 177,A 169.6867,B 6.5586,C 0.2336,E1 6.4064,E2 282.6442} C_DIS
LIN {X -134.6651,Y 32.2801,Z 177,A 168.1872,B 6.5588,C 0.2289,E1 6.4073,E2 284.1372} C_DIS
LIN {X -133.7983,Y 35.7023,Z 177,A 166.596,B 6.5588,C 0.2263,E1 6.4084,E2 285.7434} C_DIS
LIN {X -132.5053,Y 40.2377,Z 177,A 164.6407,B 6.5591,C 0.2209,E1 6.41,E2 287.6974} C_DIS
LIN {X -131.4636,Y 43.5203,Z 177,A 163.3995,B 6.5593,C 0.215,E1 6.411,E2 288.9143} C_DIS
LIN {X -129.8773,Y 48.0502,Z 177,A 161.3107,B 6.5593,C 0.2108,E1 6.413,E2 291.0143} C_DIS
LIN {X -127.6551,Y 53.6739,Z 177,A 158.6176,B 6.5595,C 0.2063,E1 6.4158,E2 293.729} C_DIS
LIN {X -126.1597,Y 57.1027,Z 177,A 157.0495,B 6.5597,C 0.2024,E1 6.4176,E2 295.2983} C_DIS
LIN {X -124.5604,Y 60.5144,Z 177,A 155.3373,B 6.5597,C 0.2001,E1 6.4196,E2 297.0281} C_DIS
LIN {X -121.5376,Y 66.3759,Z 177,A 152.6229,B 6.5599,C 0.193,E1 6.4232,E2 299.7381} C_DIS
LIN {X -119.3258,Y 70.2747,Z 177,A 150.7078,B 6.5601,C 0.1891,E1 6.4258,E2 301.659} C_DIS
LIN {X -116.9197,Y 74.2095,Z 177,A 148.7354,B 6.5601,C 0.1852,E1 6.4288,E2 303.6377} C_DIS
LIN {X -114.4033,Y 78.0333,Z 177,A 146.7853,B 6.5603,C 0.1813,E1 6.4318,E2 305.5929} C_DIS
LIN {X -111.7355,Y 81.8069,Z 177,A 144.9735,B 6.5604,C 0.1757,E1 6.4347,E2 307.3906} C_DIS
LIN {X -109.338,Y 84.9846,Z 177,A 143.2506,B 6.5604,C 0.1728,E1 6.4377,E2 309.1213} C_DIS
LIN {X -106.7936,Y 88.1607,Z 177,A 141.4756,B 6.5606,C 0.1702,E1 6.4408,E2 310.9061} C_DIS
LIN {X -103.9698,Y 91.4742,Z 177,A 139.8176,B 6.5607,C 0.1646,E1 6.4438,E2 312.5448} C_DIS
LIN {X -102.0127,Y 93.6513,Z 177,A 138.3377,B 6.5607,C 0.1652,E1 6.4466,E2 314.0567} C_DIS
LIN {X -98.6075,Y 97.2309,Z 177,A 136.3239,B 6.5608,C 0.1606,E1 6.4505,E2 316.065} C_DIS
LIN {X -95.31,Y 100.4654,Z 177,A 134.5392,B 6.5609,C 0.1553,E1 6.4541,E2 317.8324} C_DIS
LIN {X -92.463,Y 103.091,Z 177,A 132.6958,B 6.5609,C 0.1551,E1 6.458,E2 319.7041} C_DIS
LIN {X -88.6838,Y 106.3603,Z 177,A 130.6718,B 6.561,C 0.1507,E1 6.4623,E2 321.721} C_DIS
LIN {X -85.2963,Y 109.0953,Z 177,A 128.8802,B 6.5611,C 0.1474,E1 6.4662,E2 323.5098} C_DIS
LIN {X -82.1988,Y 111.4476,Z 177,A 127.1291,B 6.5611,C 0.1464,E1 6.4701,E2 325.277} C_DIS
LIN {X -78.0642,Y 114.3821,Z 177,A 125.089,B 6.5612,C 0.1423,E1 6.4748,E2 327.3083} C_DIS
LIN {X -74.2687,Y 116.8823,Z 177,A 123.1655,B 6.5612,C 0.1399,E1 6.4793,E2 329.2356} C_DIS
LIN {X -70.3951,Y 119.255,Z 177,A 121.2796,B 6.5613,C 0.1372,E1 6.4838,E2 331.1207} C_DIS
LIN {X -66.5597,Y 121.4374,Z 177,A 119.4539,B 6.5613,C 0.1347,E1 6.4883,E2 332.945} C_DIS
LIN {X -63.1926,Y 123.2212,Z 177,A 118.0475,B 6.5615,C 0.1304,E1 6.4917,E2 334.3292} C_DIS
LIN {X -58.7511,Y 125.4009,Z 177,A 115.7845,B 6.5615,C 0.1307,E1 6.4974,E2 336.6173} C_DIS
LIN {X -55.0424,Y 127.0706,Z 177,A 113.5374,B 6.5614,C 0.136,E1 6.5034,E2 338.9321} C_DIS
LIN {X -50.2447,Y 129.043,Z 177,A 112.1006,B 6.5616,C 0.1246,E1 6.5069,E2 340.2806} C_DIS
LIN {X -47.213,Y 130.183,Z 177,A 110.7132,B 6.5616,C 0.1239,E1 6.5105,E2 341.6729} C_DIS
LIN {X -44.0405,Y 131.2904,Z 177,A 109.2333,B 6.5616,C 0.1238,E1 6.5144,E2 343.1629} C_DIS
LIN {X -40.7637,Y 132.3443,Z 177,A 107.8397,B 6.5616,C 0.1222,E1 6.5181,E2 344.5518} C_DIS
LIN {X -37.8649,Y 133.2038,Z 177,A 106.5804,B 6.5616,C 0.1213,E1 6.5215,E2 345.8113} C_DIS
LIN {X -34.7621,Y 134.0476,Z 177,A 105.1722,B 6.5616,C 0.1213,E1 6.5254,E2 347.2282} C_DIS
LIN {X -31.0387,Y 134.9567,Z 177,A 103.6337,B 6.5616,C 0.1197,E1 6.5295,E2 348.76} C_DIS
LIN {X -27.6472,Y 135.692,Z 177,A 102.1857,B 6.5616,C 0.119,E1 6.5335,E2 350.2086} C_DIS
LIN {X -23.719,Y 136.4352,Z 177,A 100.5889,B 6.5617,C 0.1175,E1 6.5378,E2 351.7974} C_DIS
LIN {X -19.7897,Y 137.0588,Z 177,A 98.9244,B 6.5617,C 0.117,E1 6.5424,E2 353.4632} C_DIS
LIN {X -11.1778,Y 138.029,Z 177,A 95.3198,B 6.5617,C 0.1163,E1 6.5525,E2 357.0685} C_DIS
LIN {X -6.1657,Y 138.3449,Z 177,A 93.0802,B 6.5617,C 0.1182,E1 6.5587,E2 359.3269} C_DIS
LIN {X -2.3919,Y 138.4595,Z 177,A 91.671,B 6.5617,C 0.116,E1 6.5626,E2 360.7165} C_DIS
LIN {X 1.437,Y 138.4743,Z 177,A 89.9865,B 6.5617,C 0.1174,E1 6.5674,E2 362.4128} C_DIS
LIN {X 5.2421,Y 138.381,Z 177,A 88.4798,B 6.5617,C 0.1166,E1 6.5715,E2 363.9103} C_DIS
LIN {X 8.8752,Y 138.1958,Z 177,A 86.9258,B 6.5617,C 0.1176,E1 6.5759,E2 365.4697} C_DIS
LIN {X 12.9235,Y 137.876,Z 177,A 84.9003,B 6.5617,C 0.123,E1 6.5817,E2 367.537} C_DIS
LIN {X 16.9087,Y 137.4448,Z 177,A 83.3111,B 6.5617,C 0.1226,E1 6.586,E2 369.1172} C_DIS
LIN {X 20.5371,Y 136.9502,Z 177,A 82.0668,B 6.5617,C 0.1194,E1 6.5894,E2 370.3278} C_DIS
LIN {X 24.1165,Y 136.3641,Z 177,A 80.7927,B 6.5617,C 0.1168,E1 6.5928,E2 371.5734} C_DIS
LIN {X 29.9452,Y 135.2054,Z 177,A 78.1799,B 6.5617,C 0.1205,E1 6.6,E2 374.2047} C_DIS
LIN {X 34.8001,Y 134.038,Z 177,A 76.0821,B 6.5617,C 0.1224,E1 6.6057,E2 376.3059} C_DIS
LIN {X 38.6085,Y 132.9892,Z 177,A 74.5141,B 6.5617,C 0.1227,E1 6.6099,E2 377.8653} C_DIS
LIN {X 41.8219,Y 132.0139,Z 177,A 73.1088,B 6.5616,C 0.1242,E1 6.6136,E2 379.2723} C_DIS
LIN {X 45.0617,Y 130.9434,Z 177,A 71.7688,B 6.5616,C 0.1244,E1 6.6172,E2 380.6032} C_DIS
LIN {X 48.1164,Y 129.8525,Z 177,A 70.3926,B 6.5616,C 0.1262,E1 6.6208,E2 381.9835} C_DIS
LIN {X 51.6232,Y 128.4978,Z 177,A 68.9665,B 6.5616,C 0.1259,E1 6.6245,E2 383.3933} C_DIS
LIN {X 55.8695,Y 126.7112,Z 177,A 66.1932,B 6.5612,C 0.1414,E1 6.6318,E2 386.2732} C_DIS
LIN {X 61.2621,Y 124.1916,Z 177,A 64.5832,B 6.5615,C 0.1313,E1 6.6356,E2 387.7782} C_DIS
LIN {X 63.8352,Y 122.8903,Z 177,A 63.2879,B 6.5614,C 0.1345,E1 6.6389,E2 389.0862} C_DIS
LIN {X 67.6815,Y 120.8156,Z 177,A 61.4621,B 6.5614,C 0.1373,E1 6.6433,E2 390.9142} C_DIS
LIN {X 71.8276,Y 118.3976,Z 177,A 59.3986,B 6.5612,C 0.1414,E1 6.6483,E2 392.9874} C_DIS
LIN {X 74.7109,Y 116.5995,Z 177,A 57.3729,B 6.561,C 0.1534,E1 6.6533,E2 395.0895} C_DIS
LIN {X 80.0092,Y 113.0297,Z 177,A 55.5161,B 6.5612,C 0.1453,E1 6.6573,E2 396.8497} C_DIS
LIN {X 83.6127,Y 110.3907,Z 177,A 53.7071,B 6.5612,C 0.1478,E1 6.6613,E2 398.6541} C_DIS
LIN {X 86.8164,Y 107.8892,Z 177,A 52.0334,B 6.561,C 0.1507,E1 6.665,E2 400.327} C_DIS
LIN {X 90.2863,Y 105.0025,Z 177,A 50.1995,B 6.561,C 0.1536,E1 6.6689,E2 402.1571} C_DIS
LIN {X 93.481,Y 102.1692,Z 177,A 48.6622,B 6.561,C 0.1532,E1 6.672,E2 403.6662} C_DIS
LIN {X 95.6221,Y 100.1677,Z 177,A 47.15,B 6.5608,C 0.1605,E1 6.6752,E2 405.2159} C_DIS
LIN {X 99.2442,Y 96.5809,Z 177,A 45.1492,B 6.5608,C 0.163,E1 6.6791,E2 407.2039} C_DIS
LIN {X 102.4675,Y 93.1535,Z 177,A 43.2839,B 6.5607,C 0.1657,E1 6.6826,E2 409.0596} C_DIS
LIN {X 105.1953,Y 90.0625,Z 177,A 41.6114,B 6.5607,C 0.1689,E1 6.6857,E2 410.7284} C_DIS
LIN {X 108.0247,Y 86.6484,Z 177,A 39.8788,B 6.5605,C 0.1712,E1 6.6887,E2 412.449} C_DIS
LIN {X 110.8654,Y 82.9826,Z 177,A 37.8639,B 6.5604,C 0.1772,E1 6.6921,E2 414.4766} C_DIS
LIN {X 113.5353,Y 79.2903,Z 177,A 36.0322,B 6.5603,C 0.1807,E1 6.6951,E2 416.3023} C_DIS
LIN {X 116.5647,Y 74.7652,Z 177,A 32.5699,B 6.5595,C 0.2064,E1 6.7006,E2 419.9153} C_DIS
LIN {X 121.2979,Y 66.8136,Z 177,A 30.0946,B 6.5599,C 0.1931,E1 6.7037,E2 422.2247} C_DIS
LIN {X 123.1989,Y 63.2362,Z 177,A 28.4634,B 6.5599,C 0.1965,E1 6.7058,E2 423.8512} C_DIS
LIN {X 124.9571,Y 59.685,Z 177,A 26.6823,B 6.5596,C 0.2032,E1 6.708,E2 425.6509} C_DIS
LIN {X 126.777,Y 55.7215,Z 177,A 23.9651,B 6.559,C 0.2235,E1 6.7112,E2 428.4827} C_DIS
LIN {X 129.8708,Y 48.0674,Z 177,A 21.6873,B 6.5593,C 0.2131,E1 6.7133,E2 430.6209} C_DIS
LIN {X 131.294,Y 44.0296,Z 177,A 20.019,B 6.5593,C 0.2161,E1 6.7148,E2 432.2772} C_DIS
LIN {X 132.3874,Y 40.6228,Z 177,A 18.5741,B 6.5591,C 0.2195,E1 6.716,E2 433.7186} C_DIS
LIN {X 133.4944,Y 36.8258,Z 177,A 16.904,B 6.5589,C 0.2246,E1 6.7173,E2 435.3941} C_DIS
LIN {X 134.5517,Y 32.7504,Z 177,A 15.2511,B 6.5589,C 0.2279,E1 6.7184,E2 437.0369} C_DIS
LIN {X 135.2844,Y 29.5794,Z 177,A 13.6118,B 6.5585,C 0.2367,E1 6.7194,E2 438.7141} C_DIS
LIN {X 136.0466,Y 25.8463,Z 177,A 12.4679,B 6.5586,C 0.2336,E1 6.72,E2 439.8045} C_DIS
LIN {X 136.6838,Y 22.2384,Z 177,A 11.0207,B 6.5586,C 0.2367,E1 6.7207,E2 441.2441} C_DIS
LIN {X 137.2904,Y 18.1128,Z 177,A 8.7052,B 6.558,C 0.2519,E1 6.7216,E2 443.6355} C_DIS
LIN {X 137.8459,Y 13.2375,Z 177,A 7.3206,B 6.5582,C 0.2464,E1 6.7219,E2 444.94} C_DIS
LIN {X 138.1341,Y 9.7864,Z 177,A 5.8092,B 6.558,C 0.2518,E1 6.7223,E2 446.4625} C_DIS
LIN {X 138.3722,Y 5.4653,Z 177,A 4.0664,B 6.5578,C 0.2561,E1 6.7225,E2 448.2006} C_DIS
LIN {X 138.4786,Y 0.8377,Z 177,A 2.1858,B 6.5576,C 0.261,E1 6.7225,E2 450.0784} C_DIS
LIN {X 138.4386,Y -3.4182,Z 177,A 0.497,B 6.5574,C 0.2648,E1 6.7225,E2 451.7595} C_DIS
LIN {X 138.2755,Y -7.5488,Z 177,A -1.2184,B 6.5572,C 0.2698,E1 6.7223,E2 453.4769} C_DIS
LIN {X 137.7232,Y -14.4626,Z 177,A -3.9814,B 6.557,C 0.2761,E1 6.7216,E2 456.2288} C_DIS
LIN {X 137.2807,Y -18.1867,Z 177,A -5.4932,B 6.5568,C 0.2798,E1 6.7211,E2 457.7369} C_DIS
LIN {X 136.6636,Y -22.3593,Z 177,A -7.2898,B 6.5566,C 0.2857,E1 6.7203,E2 459.5416} C_DIS
LIN {X 135.8944,Y -26.6425,Z 177,A -9.0377,B 6.5564,C 0.2898,E1 6.7194,E2 461.2844} C_DIS
LIN {X 135.1032,Y -30.397,Z 177,A -10.497,B 6.5563,C 0.292,E1 6.7185,E2 462.7286} C_DIS
LIN {X 134.297,Y -33.7795,Z 177,A -11.9455,B 6.5561,C 0.2962,E1 6.7176,E2 464.1797} C_DIS
LIN {X 133.3959,Y -37.1779,Z 177,A -13.3689,B 6.5559,C 0.2997,E1 6.7165,E2 465.6004} C_DIS
LIN {X 132.0871,Y -41.5927,Z 177,A -15.1696,B 6.5558,C 0.3032,E1 6.7151,E2 467.3895} C_DIS
LIN {X 130.9402,Y -45.0709,Z 177,A -16.6822,B 6.5556,C 0.3073,E1 6.7137,E2 468.9031} C_DIS
LIN {X 129.6621,Y -48.6246,Z 177,A -18.2308,B 6.5554,C 0.3113,E1 6.7123,E2 470.4514} C_DIS
LIN {X 128.264,Y -52.2033,Z 177,A -19.8428,B 6.5552,C 0.3159,E1 6.7106,E2 472.0678} C_DIS
LIN {X 126.5853,Y -56.1511,Z 177,A -21.5818,B 6.555,C 0.32,E1 6.7086,E2 473.8037} C_DIS
LIN {X 124.0118,Y -61.6266,Z 177,A -23.9801,B 6.5548,C 0.3248,E1 6.7058,E2 476.1909} C_DIS
LIN {X 121.8527,Y -65.7964,Z 177,A -25.9426,B 6.5545,C 0.3301,E1 6.7032,E2 478.1578} C_DIS
LIN {X 119.6209,Y -69.7723,Z 177,A -27.8003,B 6.5543,C 0.3344,E1 6.7006,E2 480.0136} C_DIS
LIN {X 118.009,Y -72.464,Z 177,A -29.0695,B 6.5541,C 0.3371,E1 6.6988,E2 481.2803} C_DIS
LIN {X 115.5894,Y -76.2644,Z 177,A -30.8657,B 6.554,C 0.3405,E1 6.6961,E2 483.0695} C_DIS
LIN {X 113.1559,Y -79.8304,Z 177,A -32.6407,B 6.5538,C 0.3446,E1 6.6933,E2 484.8448} C_DIS
LIN {X 110.8652,Y -82.983,Z 177,A -34.0822,B 6.5538,C 0.3455,E1 6.6909,E2 486.2657} C_DIS
LIN {X 107.3815,Y -87.4438,Z 177,A -37.3018,B 6.5526,C 0.3659,E1 6.6851,E2 489.6002} C_DIS
LIN {X 103.1559,Y -92.3905,Z 177,A -38.9463,B 6.5533,C 0.354,E1 6.6823,E2 491.1127} C_DIS
LIN {X 98.4019,Y -97.4386,Z 177,A -42.0227,B 6.5527,C 0.3637,E1 6.6763,E2 494.2186} C_DIS
LIN {X 93.4795,Y -102.1706,Z 177,A -44.6037,B 6.5527,C 0.3654,E1 6.6711,E2 496.7706} C_DIS
LIN {X 87.8068,Y -107.0848,Z 177,A -47.591,B 6.5524,C 0.3694,E1 6.6649,E2 499.7455} C_DIS
LIN {X 85.8469,Y -108.6628,Z 177,A -49.1543,B 6.5518,C 0.3801,E1 6.6613,E2 501.3774} C_DIS
LIN {X 82.8372,Y -110.9737,Z 177,A -50.3986,B 6.5519,C 0.3775,E1 6.6586,E2 502.5809} C_DIS
LIN {X 78.0344,Y -114.4025,Z 177,A -52.8494,B 6.5517,C 0.3819,E1 6.653,E2 505.035} C_DIS
LIN {X 74.2089,Y -116.9201,Z 177,A -54.7331,B 6.5515,C 0.3849,E1 6.6485,E2 506.9189} C_DIS
LIN {X 71.1195,Y -118.8244,Z 177,A -56.1733,B 6.5515,C 0.3862,E1 6.6451,E2 508.3524} C_DIS
LIN {X 66.6632,Y -121.3809,Z 177,A -58.3181,B 6.5512,C 0.3897,E1 6.6399,E2 510.5014} C_DIS
LIN {X 63.0956,Y -123.2705,Z 177,A -59.8338,B 6.5512,C 0.3896,E1 6.6362,E2 511.9983} C_DIS
LIN {X 59.93,Y -124.8401,Z 177,A -61.2382,B 6.5512,C 0.3906,E1 6.6327,E2 513.3963} C_DIS
LIN {X 56.783,Y -126.3026,Z 177,A -62.7072,B 6.551,C 0.393,E1 6.6289,E2 514.8708} C_DIS
LIN {X 53.7862,Y -127.6082,Z 177,A -64.0263,B 6.551,C 0.3942,E1 6.6256,E2 516.1866} C_DIS
LIN {X 50.6044,Y -128.9031,Z 177,A -65.3892,B 6.551,C 0.3949,E1 6.622,E2 517.5429} C_DIS
LIN {X 47.4028,Y -130.1146,Z 177,A -66.9054,B 6.5507,C 0.3981,E1 6.618,E2 519.0732} C_DIS
LIN {X 44.0399,Y -131.2905,Z 177,A -68.3419,B 6.5507,C 0.399,E1 6.6142,E2 520.5059} C_DIS
LIN {X 40.6907,Y -132.3667,Z 177,A -69.801,B 6.5506,C 0.4005,E1 6.6104,E2 521.9664} C_DIS
LIN {X 36.9207,Y -133.4678,Z 177,A -71.4606,B 6.5505,C 0.4025,E1 6.6059,E2 523.6316} C_DIS
LIN {X 33.3995,Y -134.3934,Z 177,A -73.1377,B 6.5502,C 0.4064,E1 6.6013,E2 525.3319} C_DIS
LIN {X 28.3625,Y -135.5464,Z 177,A -75.0949,B 6.5503,C 0.4051,E1 6.596,E2 527.2671} C_DIS
LIN {X 24.6879,Y -136.2618,Z 177,A -76.5459,B 6.5503,C 0.4046,E1 6.592,E2 528.7062} C_DIS
LIN {X 16.8793,Y -137.4483,Z 177,A -79.8543,B 6.5502,C 0.407,E1 6.5829,E2 532.0218} C_DIS
LIN {X 13.4135,Y -137.829,Z 177,A -81.246,B 6.5502,C 0.4068,E1 6.579,E2 533.4077} C_DIS
LIN {X 9.3035,Y -138.1694,Z 177,A -83.0579,B 6.5501,C 0.409,E1 6.5739,E2 535.2344} C_DIS
LIN {X 5.2356,Y -138.3812,Z 177,A -84.6291,B 6.5501,C 0.4077,E1 6.5696,E2 536.7915} C_DIS
LIN {X 0.9981,Y -138.4764,Z 177,A -86.3999,B 6.5501,C 0.4082,E1 6.5646,E2 538.5654} C_DIS
Enddeposition()
LIN {X 0.9981,Y -138.4764,Z 177,A -86.3999,B 6.5501,C 0.4082,E1 6.5646,E2 538.5654} C_DIS
Startdeposition()
$VEL.CP = VEL_PRINT
LIN {X 2.3033,Y -139.3659,Z 177,A -85.2041,B 6.5556,C 0.402,E1 6.5732,E2 537.3143} C_DIS
LIN {X 6.175,Y -139.25,Z 177,A -83.4739,B 6.5558,C 0.3995,E1 6.5781,E2 535.5651} C_DIS
LIN {X 10.1789,Y -139.0127,Z 177,A -81.9128,B 6.5558,C 0.4003,E1 6.5824,E2 534.0147} C_DIS
LIN {X 13.8818,Y -138.693,Z 177,A -80.4442,B 6.5557,C 0.4007,E1 6.5865,E2 532.5531} C_DIS
LIN {X 17.2019,Y -138.321,Z 177,A -78.963,B 6.5558,C 0.3984,E1 6.5907,E2 531.0569} C_DIS
LIN {X 23.5392,Y -137.384,Z 177,A -75.7541,B 6.5565,C 0.3877,E1 6.5997,E2 527.7696} C_DIS
LIN {X 28.9217,Y -136.352,Z 177,A -74.3242,B 6.5558,C 0.3993,E1 6.6033,E2 526.4479} C_DIS
LIN {X 34.6422,Y -135.0115,Z 177,A -71.7114,B 6.5561,C 0.3942,E1 6.6105,E2 523.8075} C_DIS
LIN {X 39.8914,Y -133.5563,Z 177,A -69.5892,B 6.5561,C 0.3942,E1 6.6162,E2 521.6993} C_DIS
LIN {X 42.6326,Y -132.7048,Z 177,A -68.388,B 6.5561,C 0.3926,E1 6.6194,E2 520.4944} C_DIS
LIN {X 45.9401,Y -131.5965,Z 177,A -66.9688,B 6.5562,C 0.3914,E1 6.6231,E2 519.0762} C_DIS
LIN {X 49.1397,Y -130.4354,Z 177,A -65.5475,B 6.5564,C 0.3894,E1 6.6269,E2 517.6509} C_DIS
LIN {X 52.7526,Y -129.0181,Z 177,A -64.009,B 6.5564,C 0.3885,E1 6.6308,E2 516.1188} C_DIS
LIN {X 55.7985,Y -127.7294,Z 177,A -62.6605,B 6.5565,C 0.387,E1 6.6343,E2 514.7706} C_DIS
LIN {X 58.9106,Y -126.3239,Z 177,A -61.2735,B 6.5565,C 0.3854,E1 6.6378,E2 513.3848} C_DIS
LIN {X 61.8925,Y -124.8895,Z 177,A -59.8923,B 6.5567,C 0.3832,E1 6.6413,E2 511.9997} C_DIS
LIN {X 65.1313,Y -123.2317,Z 177,A -58.409,B 6.5568,C 0.3813,E1 6.645,E2 510.5169} C_DIS
LIN {X 71.3703,Y -119.7282,Z 177,A -55.6412,B 6.5569,C 0.3798,E1 6.6516,E2 507.7698} C_DIS
LIN {X 74.7375,Y -117.6564,Z 177,A -54.005,B 6.5571,C 0.377,E1 6.6555,E2 506.1308} C_DIS
LIN {X 77.7269,Y -115.7033,Z 177,A -52.0638,B 6.5577,C 0.3665,E1 6.6602,E2 504.1256} C_DIS
LIN {X 81.0345,Y -113.4104,Z 177,A -50.8471,B 6.5574,C 0.3711,E1 6.6628,E2 502.9656} C_DIS
LIN {X 83.2233,Y -111.8143,Z 177,A -49.5019,B 6.5578,C 0.3651,E1 6.6659,E2 501.5887} C_DIS
LIN {X 87.3414,Y -108.6281,Z 177,A -47.5744,B 6.5578,C 0.3648,E1 6.6701,E2 499.6876} C_DIS
LIN {X 92.6502,Y -104.1373,Z 177,A -44.6599,B 6.5581,C 0.3583,E1 6.6763,E2 496.7632} C_DIS
LIN {X 96.4082,Y -100.6679,Z 177,A -42.7051,B 6.5582,C 0.3565,E1 6.6802,E2 494.826} C_DIS
LIN {X 99.5425,Y -97.5697,Z 177,A -40.4852,B 6.5588,C 0.3456,E1 6.6847,E2 492.5502} C_DIS
LIN {X 102.6191,Y -94.3285,Z 177,A -39.0554,B 6.5586,C 0.3487,E1 6.6873,E2 491.1728} C_DIS
LIN {X 106.1661,Y -90.3178,Z 177,A -37.1243,B 6.5586,C 0.3486,E1 6.6908,E2 489.2753} C_DIS
LIN {X 108.2962,Y -87.753,Z 177,A -34.7942,B 6.5597,C 0.3285,E1 6.6951,E2 486.8166} C_DIS
LIN {X 112.302,Y -82.564,Z 177,A -32.8991,B 6.5593,C 0.3363,E1 6.6981,E2 485.0253} C_DIS
LIN {X 114.4463,Y -79.5651,Z 177,A -31.4385,B 6.5594,C 0.3337,E1 6.7004,E2 483.5705} C_DIS
LIN {X 117.0025,Y -75.7562,Z 177,A -29.3211,B 6.5599,C 0.3249,E1 6.7037,E2 481.4207} C_DIS
LIN {X 118.9785,Y -72.6139,Z 177,A -28.3438,B 6.5596,C 0.3309,E1 6.705,E2 480.5143} C_DIS
LIN {X 121.6575,Y -68.0302,Z 177,A -25.9418,B 6.56,C 0.3215,E1 6.7084,E2 478.0814} C_DIS
LIN {X 123.9317,Y -63.7911,Z 177,A -23.9918,B 6.5603,C 0.3169,E1 6.7109,E2 476.1331} C_DIS
LIN {X 125.9848,Y -59.6328,Z 177,A -22.2393,B 6.5603,C 0.3146,E1 6.7131,E2 474.399} C_DIS
LIN {X 127.4757,Y -56.3763,Z 177,A -20.7679,B 6.5605,C 0.3108,E1 6.7147,E2 472.9264} C_DIS
LIN {X 128.7788,Y -53.331,Z 177,A -19.4454,B 6.5607,C 0.3078,E1 6.7162,E2 471.6077} C_DIS
LIN {X 130.049,Y -50.1538,Z 177,A -18.0887,B 6.5608,C 0.3049,E1 6.7175,E2 470.2562} C_DIS
LIN {X 131.2319,Y -46.9714,Z 177,A -16.7061,B 6.561,C 0.3013,E1 6.7189,E2 468.874} C_DIS
LIN {X 132.3529,Y -43.7134,Z 177,A -15.3115,B 6.5611,C 0.2978,E1 6.7201,E2 467.481} C_DIS
LIN {X 134.3029,Y -37.2942,Z 177,A -12.6397,B 6.5614,C 0.2918,E1 6.7222,E2 464.8179} C_DIS
LIN {X 135.2367,Y -33.755,Z 177,A -11.1884,B 6.5616,C 0.2885,E1 6.7232,E2 463.3722} C_DIS
LIN {X 135.9272,Y -30.8528,Z 177,A -9.9336,B 6.5617,C 0.2846,E1 6.724,E2 462.1126} C_DIS
LIN {X 136.7041,Y -27.2108,Z 177,A -8.3837,B 6.5619,C 0.2799,E1 6.7249,E2 460.5588} C_DIS
LIN {X 137.3375,Y -23.8121,Z 177,A -7.0903,B 6.5619,C 0.2782,E1 6.7255,E2 459.281} C_DIS
LIN {X 137.837,Y -20.7226,Z 177,A -5.9036,B 6.5621,C 0.2763,E1 6.726,E2 458.1061} C_DIS
LIN {X 138.4447,Y -16.165,Z 177,A -3.9422,B 6.5624,C 0.2696,E1 6.7267,E2 456.1337} C_DIS
LIN {X 138.8975,Y -11.6456,Z 177,A -2.1478,B 6.5625,C 0.2656,E1 6.7272,E2 454.3471} C_DIS
LIN {X 139.1472,Y -8.1472,Z 177,A -0.6251,B 6.5627,C 0.26,E1 6.7275,E2 452.8127} C_DIS
LIN {X 139.3407,Y -3.5281,Z 177,A 1.145,B 6.5629,C 0.2569,E1 6.7276,E2 451.058} C_DIS
LIN {X 139.3869,Y 0.3165,Z 177,A 2.801,B 6.5631,C 0.251,E1 6.7276,E2 449.3909} C_DIS
LIN {X 139.3235,Y 4.1451,Z 177,A 4.2353,B 6.5631,C 0.249,E1 6.7276,E2 447.9735} C_DIS
LIN {X 139.1531,Y 8.0513,Z 177,A 5.9348,B 6.5634,C 0.2428,E1 6.7273,E2 446.2608} C_DIS
LIN {X 138.8235,Y 12.5211,Z 177,A 7.5882,B 6.5634,C 0.2409,E1 6.727,E2 444.6304} C_DIS
LIN {X 138.4754,Y 15.9071,Z 177,A 9.3866,B 6.5639,C 0.2298,E1 6.7264,E2 442.779} C_DIS
LIN {X 137.9726,Y 19.7903,Z 177,A 11.1326,B 6.5641,C 0.2227,E1 6.7257,E2 441.0139} C_DIS
LIN {X 137.1786,Y 24.7009,Z 177,A 12.5302,B 6.5639,C 0.2286,E1 6.725,E2 439.6991} C_DIS
LIN {X 136.3383,Y 28.9853,Z 177,A 14.4895,B 6.5642,C 0.2206,E1 6.7239,E2 437.7172} C_DIS
LIN {X 135.4753,Y 32.78,Z 177,A 15.8803,B 6.5642,C 0.2199,E1 6.723,E2 436.3524} C_DIS
LIN {X 134.6694,Y 35.9474,Z 177,A 17.2026,B 6.5643,C 0.2166,E1 6.7221,E2 435.0318} C_DIS
LIN {X 133.7381,Y 39.2704,Z 177,A 18.5944,B 6.5644,C 0.2131,E1 6.721,E2 433.6426} C_DIS
LIN {X 132.6622,Y 42.7659,Z 177,A 20.0375,B 6.5645,C 0.2101,E1 6.7198,E2 432.2063} C_DIS
LIN {X 131.478,Y 46.2819,Z 177,A 21.6836,B 6.5647,C 0.2039,E1 6.7183,E2 430.5437} C_DIS
LIN {X 129.3817,Y 51.8504,Z 177,A 24.3732,B 6.565,C 0.193,E1 6.7156,E2 427.8211} C_DIS
LIN {X 127.7877,Y 55.6637,Z 177,A 25.5933,B 6.565,C 0.197,E1 6.7143,E2 426.6619} C_DIS
LIN {X 126.4882,Y 58.5554,Z 177,A 26.9906,B 6.565,C 0.192,E1 6.7126,E2 425.2517} C_DIS
LIN {X 124.9575,Y 61.7547,Z 177,A 28.3499,B 6.5651,C 0.19,E1 6.711,E2 423.9043} C_DIS
LIN {X 123.1586,Y 65.2704,Z 177,A 29.9226,B 6.5652,C 0.1867,E1 6.709,E2 422.3373} C_DIS
LIN {X 120.5851,Y 69.9127,Z 177,A 32.4965,B 6.5656,C 0.1745,E1 6.7053,E2 419.7119} C_DIS
LIN {X 118.4118,Y 73.5338,Z 177,A 33.6564,B 6.5654,C 0.1803,E1 6.7038,E2 418.6253} C_DIS
LIN {X 116.6306,Y 76.3283,Z 177,A 35.2285,B 6.5656,C 0.1734,E1 6.7013,E2 417.0257} C_DIS
LIN {X 113.9741,Y 80.2402,Z 177,A 37.0903,B 6.5656,C 0.1702,E1 6.6984,E2 415.1737} C_DIS
LIN {X 111.3214,Y 83.8815,Z 177,A 39.3872,B 6.566,C 0.1583,E1 6.6944,E2 412.8189} C_DIS
LIN {X 108.3021,Y 87.7457,Z 177,A 40.7866,B 6.5658,C 0.1644,E1 6.6921,E2 411.4979} C_DIS
LIN {X 105.9189,Y 90.6086,Z 177,A 42.4267,B 6.5659,C 0.1592,E1 6.6891,E2 409.8434} C_DIS
LIN {X 102.9024,Y 94.0204,Z 177,A 44.284,B 6.566,C 0.1555,E1 6.6857,E2 407.9874} C_DIS
LIN {X 99.784,Y 97.3234,Z 177,A 46.1138,B 6.5661,C 0.1523,E1 6.6821,E2 406.1619} C_DIS
LIN {X 94.6334,Y 102.3388,Z 177,A 48.8451,B 6.5661,C 0.1502,E1 6.6767,E2 403.4584} C_DIS
LIN {X 91.3503,Y 105.2797,Z 177,A 50.7665,B 6.5663,C 0.1449,E1 6.6726,E2 401.5228} C_DIS
LIN {X 87.9347,Y 108.1488,Z 177,A 52.5989,B 6.5663,C 0.1416,E1 6.6687,E2 399.6902} C_DIS
LIN {X 84.3087,Y 110.9991,Z 177,A 54.4792,B 6.5664,C 0.1385,E1 6.6645,E2 397.8116} C_DIS
LIN {X 80.768,Y 113.6012,Z 177,A 56.3142,B 6.5664,C 0.135,E1 6.6604,E2 395.9728} C_DIS
LIN {X 76.0508,Y 116.8113,Z 177,A 58.2182,B 6.5664,C 0.1384,E1 6.6561,E2 394.1245} C_DIS
LIN {X 71.7611,Y 119.4951,Z 177,A 60.6159,B 6.5666,C 0.1302,E1 6.6503,E2 391.6865} C_DIS
LIN {X 67.8808,Y 121.7413,Z 177,A 62.4737,B 6.5666,C 0.1273,E1 6.6458,E2 389.8269} C_DIS
LIN {X 63.1302,Y 124.2682,Z 177,A 64.4982,B 6.5666,C 0.1273,E1 6.6408,E2 387.8261} C_DIS
LIN {X 57.914,Y 126.7848,Z 177,A 66.8541,B 6.5666,C 0.1248,E1 6.6349,E2 385.4736} C_DIS
LIN {X 55.3622,Y 127.9181,Z 177,A 68.1632,B 6.5668,C 0.1209,E1 6.6315,E2 384.1441} C_DIS
LIN {X 51.7681,Y 129.4149,Z 177,A 69.619,B 6.5668,C 0.1215,E1 6.6278,E2 382.7067} C_DIS
LIN {X 48.4068,Y 130.7099,Z 177,A 71.0687,B 6.5668,C 0.1204,E1 6.624,E2 381.2613} C_DIS
LIN {X 45.054,Y 131.9037,Z 177,A 72.5052,B 6.5668,C 0.1194,E1 6.6202,E2 379.8283} C_DIS
LIN {X 41.6821,Y 133.0084,Z 177,A 73.9697,B 6.5668,C 0.1181,E1 6.6163,E2 378.3633} C_DIS
LIN {X 38.836,Y 133.8654,Z 177,A 75.1772,B 6.5668,C 0.1173,E1 6.6131,E2 377.1579} C_DIS
LIN {X 35.2821,Y 134.8468,Z 177,A 77.06,B 6.5669,C 0.1105,E1 6.6079,E2 375.2289} C_DIS
LIN {X 31.6983,Y 135.7341,Z 177,A 78.1479,B 6.5669,C 0.116,E1 6.6051,E2 374.1958} C_DIS
LIN {X 25.8332,Y 136.9703,Z 177,A 80.7701,B 6.5669,C 0.1122,E1 6.5979,E2 371.5543} C_DIS
LIN {X 18.9,Y 138.0993,Z 177,A 83.7619,B 6.5669,C 0.1094,E1 6.5896,E2 368.5504} C_DIS
LIN {X 13.743,Y 138.7063,Z 177,A 85.7763,B 6.5669,C 0.1104,E1 6.584,E2 366.5519} C_DIS
LIN {X 9.3368,Y 139.0739,Z 177,A 87.4658,B 6.5669,C 0.1119,E1 6.5794,E2 364.8793} C_DIS
LIN {X 5.5479,Y 139.2745,Z 177,A 89.0625,B 6.5669,C 0.1111,E1 6.5749,E2 363.2784} C_DIS
LIN {X 1.9871,Y 139.3712,Z 177,A 90.5418,B 6.5669,C 0.1108,E1 6.5707,E2 361.7978} C_DIS
LIN {X -2.1486,Y 139.3685,Z 177,A 92.2095,B 6.5669,C 0.1113,E1 6.5661,E2 360.135} C_DIS
LIN {X -5.5429,Y 139.2747,Z 177,A 93.6375,B 6.5669,C 0.1109,E1 6.5621,E2 358.7036} C_DIS
LIN {X -9.6927,Y 139.0482,Z 177,A 95.1693,B 6.5669,C 0.1137,E1 6.5579,E2 357.1949} C_DIS
LIN {X -16.2107,Y 138.4392,Z 177,A 97.8094,B 6.5669,C 0.1151,E1 6.5506,E2 354.5627} C_DIS
LIN {X -19.0944,Y 138.0721,Z 177,A 99.9586,B 6.5671,C 0.1022,E1 6.5443,E2 352.2939} C_DIS
LIN {X -24.7555,Y 137.1688,Z 177,A 101.6206,B 6.5669,C 0.113,E1 6.54,E2 350.721} C_DIS
LIN {X -27.913,Y 136.5612,Z 177,A 102.9117,B 6.5669,C 0.1142,E1 6.5365,E2 349.4346} C_DIS
LIN {X -31.5394,Y 135.7704,Z 177,A 104.4275,B 6.5669,C 0.1152,E1 6.5323,E2 347.921} C_DIS
LIN {X -34.9441,Y 134.9349,Z 177,A 106.149,B 6.5669,C 0.1124,E1 6.5276,E2 346.1651} C_DIS
LIN {X -39.3713,Y 133.7086,Z 177,A 107.821,B 6.5669,C 0.1168,E1 6.5232,E2 344.5215} C_DIS
LIN {X -42.5772,Y 132.7224,Z 177,A 109.1897,B 6.5669,C 0.1181,E1 6.5195,E2 343.155} C_DIS
LIN {X -46.0096,Y 131.5724,Z 177,A 110.6734,B 6.5668,C 0.1195,E1 6.5156,E2 341.6728} C_DIS
LIN {X -49.8478,Y 130.168,Z 177,A 112.896,B 6.5668,C 0.114,E1 6.5096,E2 339.3831} C_DIS
LIN {X -54.0368,Y 128.4841,Z 177,A 114.4423,B 6.5668,C 0.1201,E1 6.5058,E2 337.8772} C_DIS
LIN {X -57.2956,Y 127.0645,Z 177,A 115.798,B 6.5668,C 0.1232,E1 6.5023,E2 336.5359} C_DIS
LIN {X -62.0149,Y 124.8291,Z 177,A 117.893,B 6.5667,C 0.1265,E1 6.4971,E2 334.449} C_DIS
LIN {X -65.2261,Y 123.1819,Z 177,A 119.4069,B 6.5667,C 0.1281,E1 6.4933,E2 332.9324} C_DIS
LIN {X -69.1462,Y 121.0263,Z 177,A 121.319,B 6.5666,C 0.1297,E1 6.4886,E2 331.0126} C_DIS
LIN {X -72.9409,Y 118.7779,Z 177,A 123.1633,B 6.5666,C 0.132,E1 6.4842,E2 329.1658} C_DIS
LIN {X -76.8968,Y 116.2563,Z 177,A 125.0961,B 6.5665,C 0.1349,E1 6.4797,E2 327.2341} C_DIS
LIN {X -80.4829,Y 113.8029,Z 177,A 127.3179,B 6.5665,C 0.1323,E1 6.4745,E2 324.9587} C_DIS
LIN {X -83.9837,Y 111.2443,Z 177,A 128.8378,B 6.5665,C 0.1387,E1 6.4712,E2 323.4736} C_DIS
LIN {X -87.1481,Y 108.784,Z 177,A 130.3977,B 6.5663,C 0.1427,E1 6.4678,E2 321.9261} C_DIS
LIN {X -90.5841,Y 105.9397,Z 177,A 132.6595,B 6.5663,C 0.1408,E1 6.4629,E2 319.6118} C_DIS
LIN {X -93.8328,Y 103.0728,Z 177,A 134.5157,B 6.5663,C 0.1433,E1 6.459,E2 317.7476} C_DIS
LIN {X -97.2128,Y 99.8917,Z 177,A 135.9954,B 6.5661,C 0.1524,E1 6.4562,E2 316.3238} C_DIS
LIN {X -100.3251,Y 96.7652,Z 177,A 138.2679,B 6.5661,C 0.1504,E1 6.4516,E2 313.9948} C_DIS
LIN {X -103.3693,Y 93.5061,Z 177,A 139.8927,B 6.5661,C 0.1569,E1 6.4486,E2 312.3981} C_DIS
LIN {X -106.8969,Y 89.4519,Z 177,A 141.9586,B 6.5658,C 0.1634,E1 6.4449,E2 310.3524} C_DIS
LIN {X -109.7684,Y 85.9041,Z 177,A 144.0019,B 6.5658,C 0.1657,E1 6.4413,E2 308.2896} C_DIS
LIN {X -112.9775,Y 81.6375,Z 177,A 146.1095,B 6.5656,C 0.1718,E1 6.4379,E2 306.1951} C_DIS
LIN {X -115.4677,Y 78.0754,Z 177,A 147.9321,B 6.5656,C 0.1756,E1 6.435,E2 304.3696} C_DIS
LIN {X -117.9252,Y 74.3116,Z 177,A 149.8047,B 6.5654,C 0.1797,E1 6.4322,E2 302.4956} C_DIS
LIN {X -120.3418,Y 70.3315,Z 177,A 151.722,B 6.5653,C 0.1844,E1 6.4294,E2 300.5796} C_DIS
LIN {X -122.4839,Y 66.5306,Z 177,A 153.893,B 6.5653,C 0.1844,E1 6.4264,E2 298.3622} C_DIS
LIN {X -124.1915,Y 63.2809,Z 177,A 155.1663,B 6.5651,C 0.1911,E1 6.4249,E2 297.1203} C_DIS
LIN {X -125.8627,Y 59.8885,Z 177,A 156.6313,B 6.5649,C 0.1962,E1 6.4231,E2 295.6681} C_DIS
LIN {X -127.3914,Y 56.5649,Z 177,A 158.2364,B 6.5649,C 0.1989,E1 6.4212,E2 294.0515} C_DIS
LIN {X -129.7421,Y 50.9435,Z 177,A 160.7383,B 6.5647,C 0.2056,E1 6.4186,E2 291.5523} C_DIS
LIN {X -130.6708,Y 48.511,Z 177,A 161.9039,B 6.5647,C 0.2074,E1 6.4175,E2 290.3757} C_DIS
LIN {X -131.9037,Y 45.054,Z 177,A 163.2924,B 6.5644,C 0.2129,E1 6.4162,E2 289.0039} C_DIS
LIN {X -132.8565,Y 42.1574,Z 177,A 164.6516,B 6.5644,C 0.2151,E1 6.415,E2 287.6323} C_DIS
LIN {X -133.9276,Y 38.6235,Z 177,A 166.1861,B 6.5642,C 0.2191,E1 6.4138,E2 286.0971} C_DIS
LIN {X -134.7492,Y 35.6479,Z 177,A 167.4839,B 6.5642,C 0.2223,E1 6.4129,E2 284.7967} C_DIS
LIN {X -135.5624,Y 32.4185,Z 177,A 168.9152,B 6.564,C 0.2254,E1 6.4119,E2 283.3588} C_DIS
LIN {X -136.3468,Y 28.9458,Z 177,A 170.7859,B 6.564,C 0.2248,E1 6.4108,E2 281.4372} C_DIS
LIN {X -137.1105,Y 25.0816,Z 177,A 172.1469,B 6.5638,C 0.2323,E1 6.4101,E2 280.1108} C_DIS
LIN {X -137.6719,Y 21.7894,Z 177,A 173.4924,B 6.5636,C 0.2366,E1 6.4095,E2 278.77} C_DIS
LIN {X -138.2155,Y 18.0165,Z 177,A 175.0397,B 6.5635,C 0.2412,E1 6.4089,E2 277.2266} C_DIS
LIN {X -138.8781,Y 11.8752,Z 177,A 177.7411,B 6.5633,C 0.2466,E1 6.4082,E2 274.5066} C_DIS
LIN {X -139.2385,Y 6.4126,Z 177,A -179.9399,B 6.563,C 0.2523,E1 6.4078,E2 272.1808} C_DIS
LIN {X -139.3657,Y 2.3162,Z 177,A -177.7615,B 6.563,C 0.2514,E1 6.4077,E2 269.9401} C_DIS
LIN {X -139.3623,Y -2.5206,Z 177,A -176.277,B 6.5626,C 0.2629,E1 6.4077,E2 268.5222} C_DIS
LIN {X -139.206,Y -7.0604,Z 177,A -174.3747,B 6.5624,C 0.2678,E1 6.4079,E2 266.6169} C_DIS
LIN {X -138.9398,Y -11.1454,Z 177,A -172.1955,B 6.5624,C 0.2669,E1 6.4084,E2 264.375} C_DIS
LIN {X -138.5321,Y -15.4018,Z 177,A -170.6864,B 6.5621,C 0.2748,E1 6.4089,E2 262.8994} C_DIS
LIN {X -137.9708,Y -19.8035,Z 177,A -169.0077,B 6.5619,C 0.2816,E1 6.4095,E2 261.2407} C_DIS
LIN {X -137.4812,Y -22.9567,Z 177,A -167.6621,B 6.5617,C 0.2849,E1 6.4101,E2 259.8917} C_DIS
LIN {X -136.8649,Y -26.3843,Z 177,A -166.2191,B 6.5615,C 0.2888,E1 6.4108,E2 258.4483} C_DIS
Enddeposition()
END
